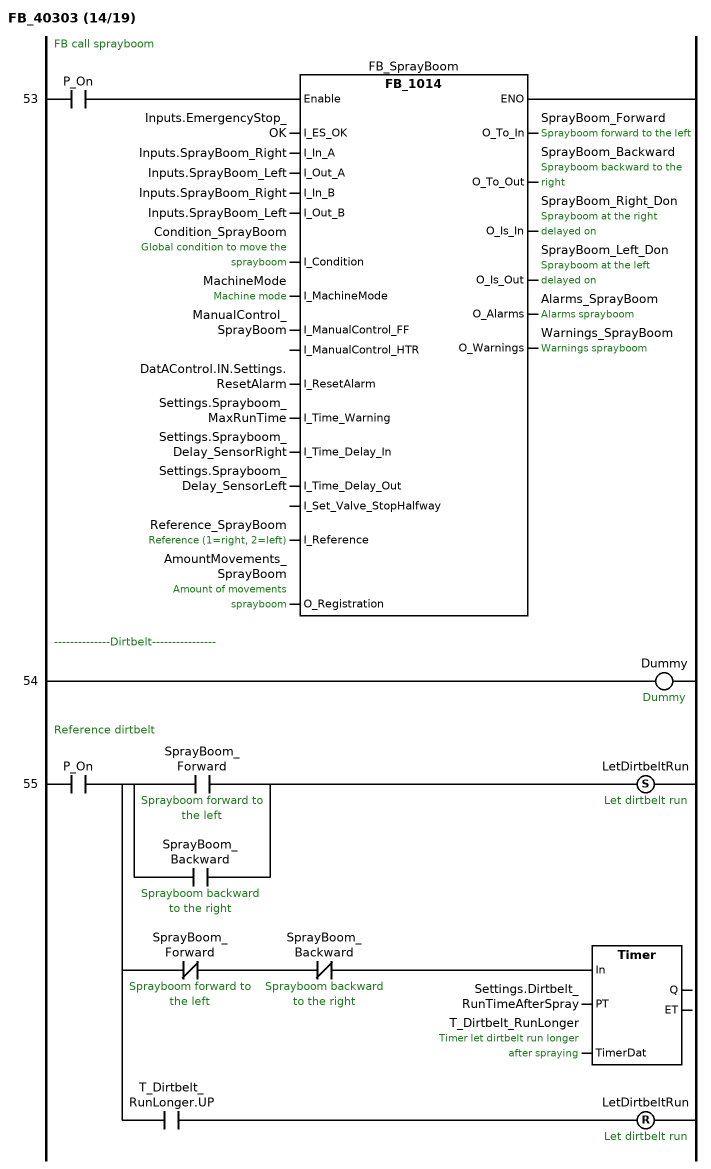
(* [picture p198: FB_40303, rungs 53-55] *)
(* Rung 53: FB call sprayboom *)
FB_SprayBoom(Enable := P_On, I_ES_OK := Inputs.EmergencyStop_OK, I_In_A := Inputs.SprayBoom_Right, I_Out_A := Inputs.SprayBoom_Left, I_In_B := Inputs.SprayBoom_Right, I_Out_B := Inputs.SprayBoom_Left, I_Condition := Condition_SprayBoom, I_MachineMode := MachineMode, I_ManualControl_FF := ManualControl_SprayBoom, I_ResetAlarm := DatAControl.IN.Settings.ResetAlarm, I_Time_Warning := Settings.Sprayboom_MaxRunTime, I_Time_Delay_In := Settings.Sprayboom_Delay_SensorRight, I_Time_Delay_Out := Settings.Sprayboom_Delay_SensorLeft, I_Reference := Reference_SprayBoom, O_Registration := AmountMovements_SprayBoom, O_To_In => SprayBoom_Forward, O_To_Out => SprayBoom_Backward, O_Is_In => SprayBoom_Right_Don, O_Is_Out => SprayBoom_Left_Don, O_Alarms => Alarms_SprayBoom, O_Warnings => Warnings_SprayBoom);
(* Rung 54: --------------Dirtbelt---------------- *)
Dummy := TRUE;
(* Rung 55: Reference dirtbelt *)
IF P_On AND (SprayBoom_Forward OR SprayBoom_Backward) THEN LetDirtbeltRun := TRUE; END_IF;
_t18 := Timer(In := P_On AND NOT SprayBoom_Forward AND NOT SprayBoom_Backward, PT := Settings.Dirtbelt_RunTimeAfterSpray, TimerDat := T_Dirtbelt_RunLonger);
IF P_On AND T_Dirtbelt_RunLonger.UP THEN LetDirtbeltRun := FALSE; END_IF;

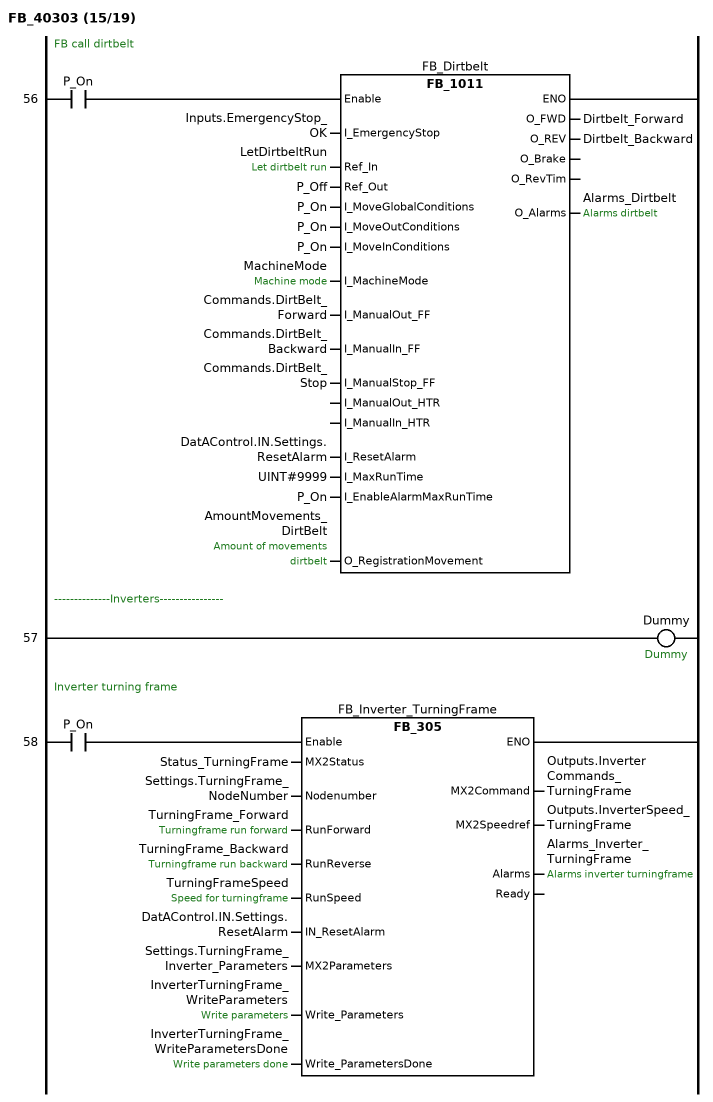
(* Rung 56: FB call dirtbelt *)
FB_Dirtbelt(Enable := P_On, I_EmergencyStop := Inputs.EmergencyStop_OK, Ref_In := LetDirtbeltRun, Ref_Out := P_Off, I_MoveGlobalConditions := P_On, I_MoveOutConditions := P_On, I_MoveInConditions := P_On, I_MachineMode := MachineMode, I_ManualOut_FF := Commands.DirtBelt_Forward, I_ManualIn_FF := Commands.DirtBelt_Backward, I_ManualStop_FF := Commands.DirtBelt_Stop, I_ResetAlarm := DatAControl.IN.Settings.ResetAlarm, I_MaxRunTime := UINT#9999, I_EnableAlarmMaxRunTime := P_On, O_RegistrationMovement := AmountMovements_DirtBelt, O_FWD => Dirtbelt_Forward, O_REV => Dirtbelt_Backward, O_Alarms => Alarms_Dirtbelt);
(* Rung 57: --------------Inverters---------------- *)
Dummy := TRUE;
(* Rung 58: Inverter turning frame *)
FB_Inverter_TurningFrame(Enable := P_On, MX2Status := Status_TurningFrame, Nodenumber := Settings.TurningFrame_NodeNumber, RunForward := TurningFrame_Forward, RunReverse := TurningFrame_Backward, RunSpeed := TurningFrameSpeed, IN_ResetAlarm := DatAControl.IN.Settings.ResetAlarm, MX2Parameters := Settings.TurningFrame_Inverter_Parameters, Write_Parameters := InverterTurningFrame_WriteParameters, Write_ParametersDone := InverterTurningFrame_WriteParametersDone, MX2Command => Outputs.InverterCommands_TurningFrame, MX2Speedref => Outputs.InverterSpeed_TurningFrame, Alarms => Alarms_Inverter_TurningFrame);

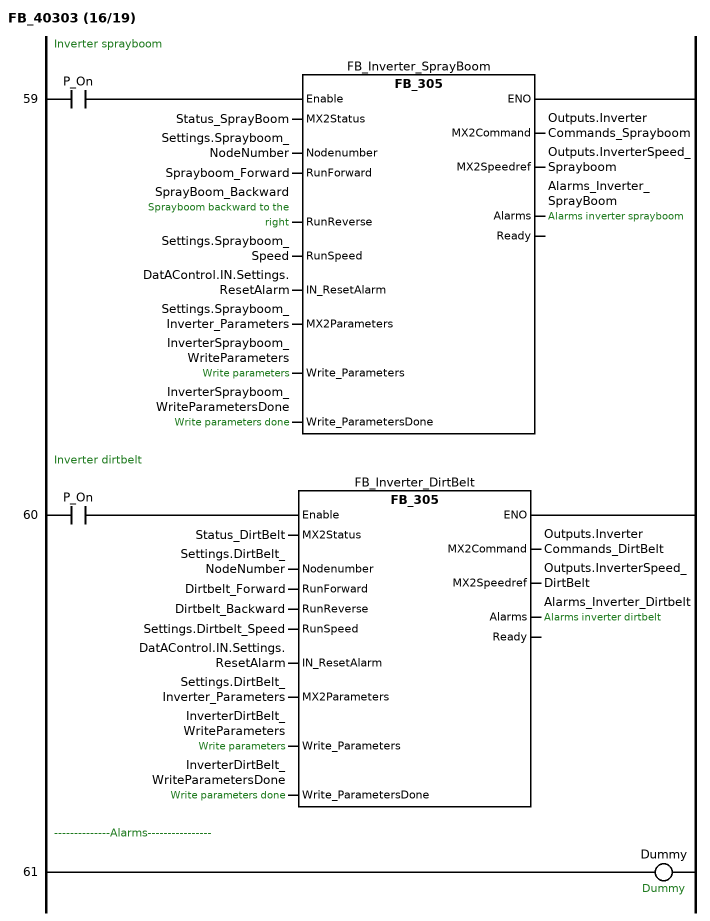
(* Rung 59: Inverter sprayboom *)
FB_Inverter_SprayBoom(Enable := P_On, MX2Status := Status_SprayBoom, Nodenumber := Settings.Sprayboom_NodeNumber, RunForward := Sprayboom_Forward, RunReverse := SprayBoom_Backward, RunSpeed := Settings.Sprayboom_Speed, IN_ResetAlarm := DatAControl.IN.Settings.ResetAlarm, MX2Parameters := Settings.Sprayboom_Inverter_Parameters, Write_Parameters := InverterSprayboom_WriteParameters, Write_ParametersDone := InverterSprayboom_WriteParametersDone, MX2Command => Outputs.InverterCommands_Sprayboom, MX2Speedref => Outputs.InverterSpeed_Sprayboom, Alarms => Alarms_Inverter_SprayBoom);
(* Rung 60: Inverter dirtbelt *)
FB_Inverter_DirtBelt(Enable := P_On, MX2Status := Status_DirtBelt, Nodenumber := Settings.DirtBelt_NodeNumber, RunForward := Dirtbelt_Forward, RunReverse := Dirtbelt_Backward, RunSpeed := Settings.Dirtbelt_Speed, IN_ResetAlarm := DatAControl.IN.Settings.ResetAlarm, MX2Parameters := Settings.DirtBelt_Inverter_Parameters, Write_Parameters := InverterDirtBelt_WriteParameters, Write_ParametersDone := InverterDirtBelt_WriteParametersDone, MX2Command => Outputs.InverterCommands_DirtBelt, MX2Speedref => Outputs.InverterSpeed_DirtBelt, Alarms => Alarms_Inverter_Dirtbelt);
(* Rung 61: --------------Alarms---------------- *)
Dummy := TRUE;

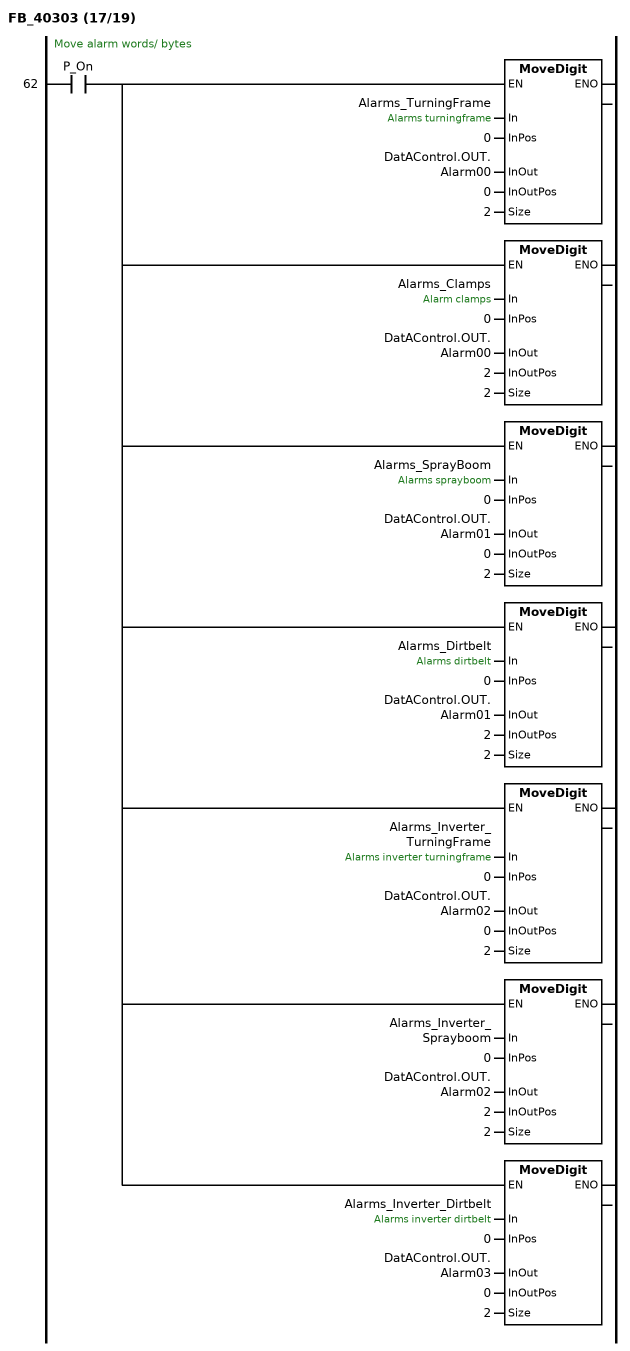
(* Rung 62: Move alarm words/ bytes *)
IF P_On THEN
    MoveDigit(In := Alarms_TurningFrame, InPos := 0, InOut := DatAControl.OUT.Alarm00, InOutPos := 0, Size := 2);
    MoveDigit(In := Alarms_Clamps, InPos := 0, InOut := DatAControl.OUT.Alarm00, InOutPos := 2, Size := 2);
    MoveDigit(In := Alarms_SprayBoom, InPos := 0, InOut := DatAControl.OUT.Alarm01, InOutPos := 0, Size := 2);
    MoveDigit(In := Alarms_Dirtbelt, InPos := 0, InOut := DatAControl.OUT.Alarm01, InOutPos := 2, Size := 2);
    MoveDigit(In := Alarms_Inverter_TurningFrame, InPos := 0, InOut := DatAControl.OUT.Alarm02, InOutPos := 0, Size := 2);
    MoveDigit(In := Alarms_Inverter_Sprayboom, InPos := 0, InOut := DatAControl.OUT.Alarm02, InOutPos := 2, Size := 2);
    MoveDigit(In := Alarms_Inverter_Dirtbelt, InPos := 0, InOut := DatAControl.OUT.Alarm03, InOutPos := 0, Size := 2);
END_IF;

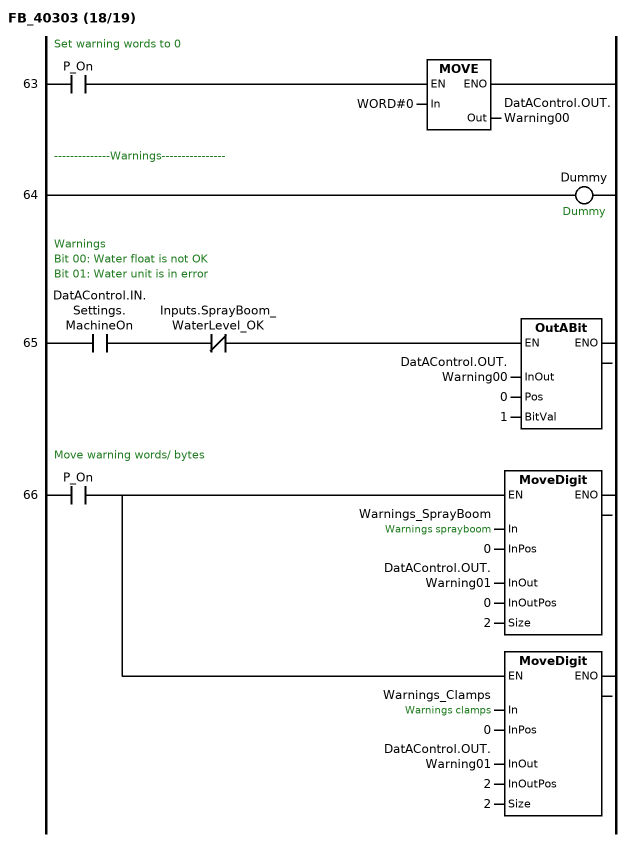
(* Rung 63: Set warning words to 0 *)
IF P_On THEN DatAControl.OUT.Warning00 := WORD#0; END_IF;
(* Rung 64: --------------Warnings---------------- *)
Dummy := TRUE;
(* Rung 65: Warnings / Bit 00: Water float is not OK / Bit 01: Water unit is in error *)
IF DatAControl.IN.Settings.MachineOn AND NOT Inputs.SprayBoom_WaterLevel_OK THEN
    OutABit(InOut := DatAControl.OUT.Warning00, Pos := 0, BitVal := 1);
END_IF;
(* Rung 66: Move warning words/ bytes *)
IF P_On THEN
    MoveDigit(In := Warnings_SprayBoom, InPos := 0, InOut := DatAControl.OUT.Warning01, InOutPos := 0, Size := 2);
    MoveDigit(In := Warnings_Clamps, InPos := 0, InOut := DatAControl.OUT.Warning01, InOutPos := 2, Size := 2);
END_IF;

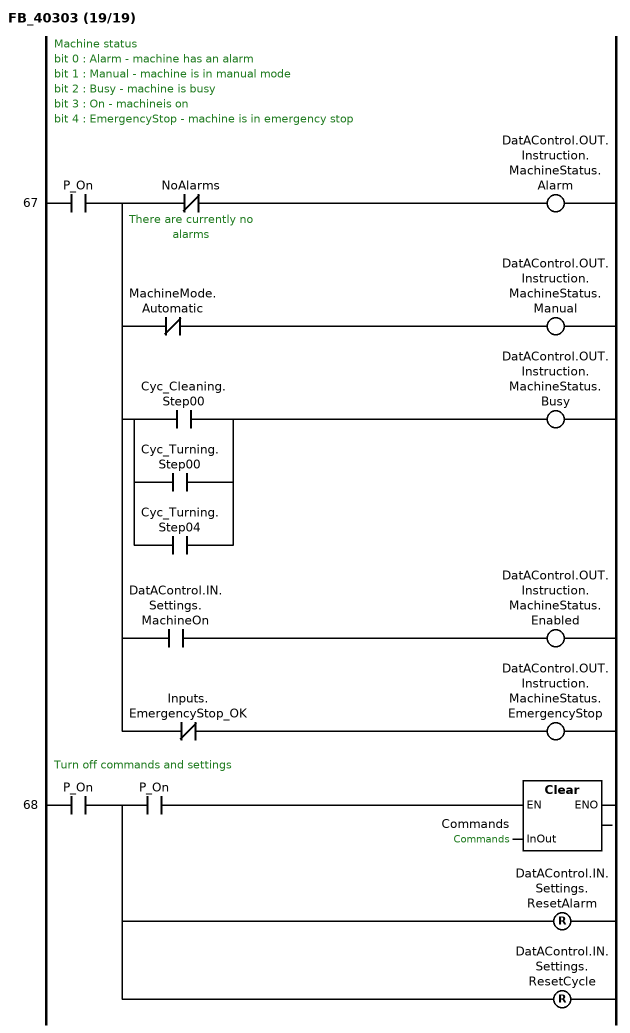
(* Rung 67: Machine status / bit 0 : Alarm - machine has an alarm / bit 1 : Manual - machine is in manual mode / bit 2 : Busy - machine is busy / bit 3 : On - machineis on / bit 4 : EmergencyStop - machine is in emergency stop *)
DatAControl.OUT.Instruction.MachineStatus.Alarm := P_On AND NOT NoAlarms;
DatAControl.OUT.Instruction.MachineStatus.Manual := P_On AND NOT MachineMode.Automatic;
DatAControl.OUT.Instruction.MachineStatus.Busy := P_On AND (Cyc_Cleaning.Step00 OR Cyc_Turning.Step00 OR Cyc_Turning.Step04);
DatAControl.OUT.Instruction.MachineStatus.Enabled := P_On AND DatAControl.IN.Settings.MachineOn;
DatAControl.OUT.Instruction.MachineStatus.EmergencyStop := P_On AND NOT Inputs.EmergencyStop_OK;
(* Rung 68: Turn off commands and settings *)
IF P_On AND P_On THEN Clear(InOut := Commands); END_IF;
IF P_On THEN
    DatAControl.IN.Settings.ResetAlarm := FALSE;
    DatAControl.IN.Settings.ResetCycle := FALSE;
END_IF;
END_FUNCTION_BLOCK

FUNCTION_BLOCK FB_1017
(* Valve movement bi-directional with 4 sensors for in detection and 4 sensors for out detection *)
VAR
    Reference_In : BOOL;  (* Reference is in *)
    Reference_Out : BOOL;  (* Reference is out *)
    Manual_In : BOOL;  (* ManualControl in *)
    Manual_Out : BOOL;  (* ManualControl out *)
    Desired_To_Out : BOOL;  (* Movement desired to Out *)
    Desired_To_In : BOOL;  (* Movement desired to In *)
    Sensor_Out_A : BOOL;  (* Sensor out side A *)
    Sensor_Out_A_Don : BOOL;  (* Sensor out side A delayed *)
    Sensor_In_A : BOOL;  (* Sensor in side A *)
    Sensor_In_A_Don : BOOL;  (* Sensor in side A delayed *)
    ManualControl : FB_303;
    Actuator_is_Out : BOOL;  (* Actuator is out *)
    Actuator_is_In : BOOL;  (* Actuator is in *)
    Input_Out_A : FB_101;
    Input_In_A : FB_101;
    Alarm_SensorTogether_A : FB_502;
    Alarm_MaxRunTime : BOOL;  (* Alarm maximum runtime actuator *)
    Alarm_Switch_Together_A : BOOL;  (* Alarm switches switched together side A *)
    Input_Out_B : FB_101;
    Sensor_Out_B : BOOL;  (* Sensor out side B *)
    Sensor_Out_B_Don : BOOL;  (* Sensor out side B delayed *)
    Input_In_B : FB_101;
    Sensor_In_B : BOOL;  (* Sensor in side B *)
    Sensor_In_B_Don : BOOL;  (* Sensor in side B delayed *)
    Alarm_SensorTogether_B : FB_502;
    Alarm_Switch_Together_B : BOOL;  (* Alarm switches switched together side B *)
    T_Warn_Out : _sTimer;
    T_Warn_In : _sTimer;
    ReversalProtection_A : FB_201;
    ReversalProtection_B : FB_201;
    NotRunning_A : BOOL;
    NotRunning_B : BOOL;
END_VAR
VAR_INPUT
    Enable : BOOL;
    I_ES_OK : BOOL;  (* IN: EmergencyStop OK *)
    I_In_A : BOOL;  (* IN: Sensor in side A *)
    I_Out_A : BOOL;  (* IN: Sensor out side A *)
    I_In_B : BOOL;  (* IN: Sensor in side B *)
    I_Out_B : BOOL;  (* IN: Sensor out side B *)
    I_Condition : BOOL;  (* IN: Global condition to move *)
    I_MachineMode : ST_MachineMode;  (* IN: Machine mode *)
    I_ManualControl : ST_ManualControl_Actuator;  (* IN: Manual control *)
    I_ResetAlarm : BOOL;  (* IN: Reset alarm *)
    I_Reference : UINT;  (* IN: Reference (1 = In, 2 = Out *)
    I_Time_Warning : UINT;  (* IN: Time for warnings 'does not reach end switch' *)
    I_Time_Delay_In : UINT;  (* IN: Time delay on in sensor *)
    I_Time_Delay_Out : UINT;  (* IN: Time delay on out sensor *)
END_VAR
VAR_OUTPUT
    O_To_In_A : BOOL;  (* OUT: Valve in A *)
    O_To_Out_A : BOOL;  (* OUT: Valve out A *)
    O_To_In_B : BOOL;  (* OUT: Valve in B *)
    O_To_Out_B : BOOL;  (* OUT: Valve out B *)
    O_Is_In : BOOL;  (* OUT: Unit is in *)
    O_Is_Out : BOOL;  (* OUT: Unit is out *)
    O_Alarms : BYTE;  (* OUT: Alarms *)
    O_Warnings : BYTE;  (* OUT: Warnings *)
END_VAR
VAR_IN_OUT
    O_Registration : UDINT;  (* OUT: Total amount of movements *)
END_VAR
VAR
    _t1 : BOOL;
    _t2 : BOOL;
    _e3 : R_TRIG;
    _e4 : R_TRIG;
END_VAR
(* ladder, written here as Structured Text *)

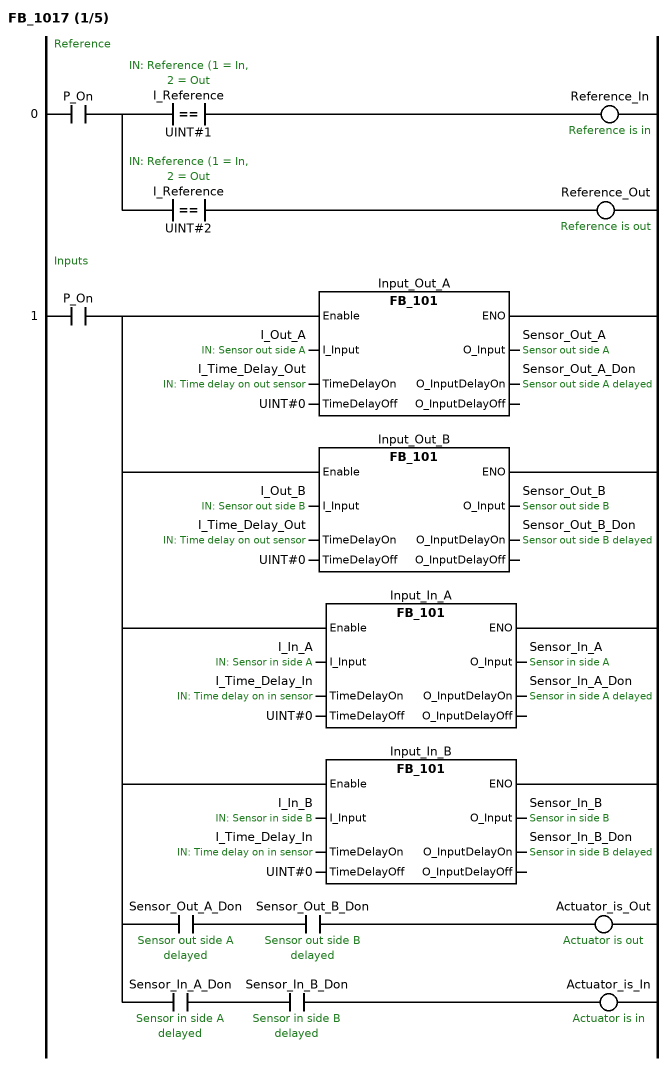
(* Rung 0: Reference *)
Reference_In := P_On AND (I_Reference = UINT#1);
Reference_Out := P_On AND (I_Reference = UINT#2);
(* Rung 1: Inputs *)
Input_Out_A(Enable := P_On, I_Input := I_Out_A, TimeDelayOn := I_Time_Delay_Out, TimeDelayOff := UINT#0, O_Input => Sensor_Out_A, O_InputDelayOn => Sensor_Out_A_Don);
Input_Out_B(Enable := P_On, I_Input := I_Out_B, TimeDelayOn := I_Time_Delay_Out, TimeDelayOff := UINT#0, O_Input => Sensor_Out_B, O_InputDelayOn => Sensor_Out_B_Don);
Input_In_A(Enable := P_On, I_Input := I_In_A, TimeDelayOn := I_Time_Delay_In, TimeDelayOff := UINT#0, O_Input => Sensor_In_A, O_InputDelayOn => Sensor_In_A_Don);
Input_In_B(Enable := P_On, I_Input := I_In_B, TimeDelayOn := I_Time_Delay_In, TimeDelayOff := UINT#0, O_Input => Sensor_In_B, O_InputDelayOn => Sensor_In_B_Don);
Actuator_is_Out := P_On AND Sensor_Out_A_Don AND Sensor_Out_B_Don;
Actuator_is_In := P_On AND Sensor_In_A_Don AND Sensor_In_B_Don;

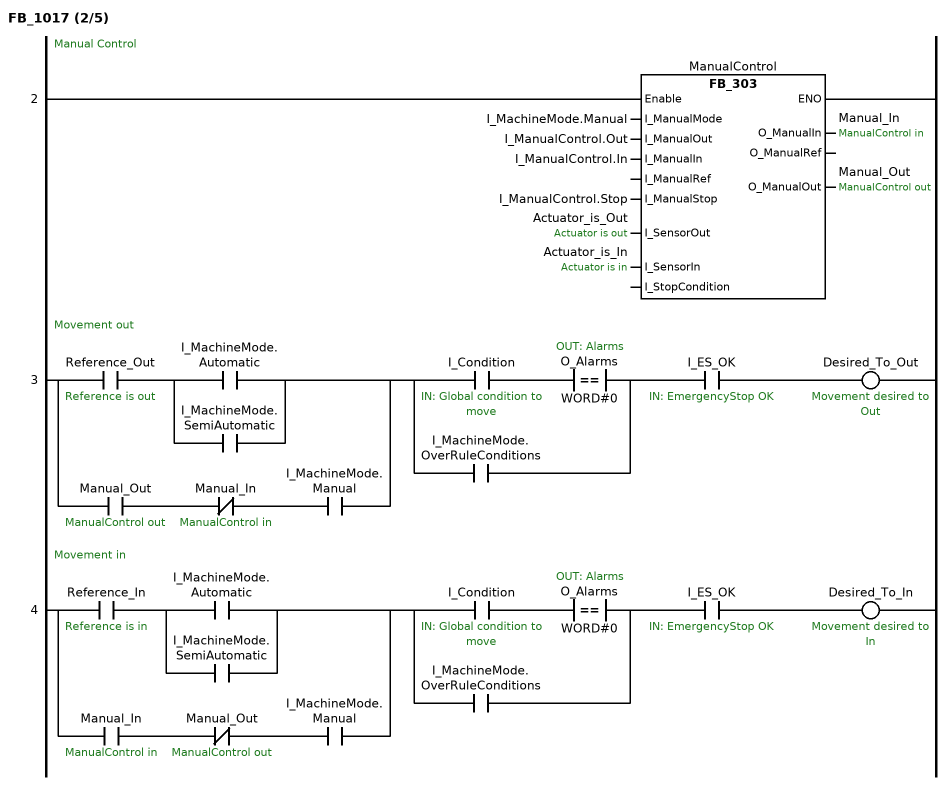
(* Rung 2: Manual Control *)
ManualControl(Enable := TRUE, I_ManualMode := I_MachineMode.Manual, I_ManualOut := I_ManualControl.Out, I_ManualIn := I_ManualControl.In, I_ManualStop := I_ManualControl.Stop, I_SensorOut := Actuator_is_Out, I_SensorIn := Actuator_is_In, O_ManualIn => Manual_In, O_ManualOut => Manual_Out);
(* Rung 3: Movement out *)
Desired_To_Out := ((Reference_Out AND (I_MachineMode.Automatic OR I_MachineMode.SemiAutomatic)) OR (Manual_Out AND NOT Manual_In AND I_MachineMode.Manual)) AND ((I_Condition AND (O_Alarms = WORD#0)) OR I_MachineMode.OverRuleConditions) AND I_ES_OK;
(* Rung 4: Movement in *)
Desired_To_In := ((Reference_In AND (I_MachineMode.Automatic OR I_MachineMode.SemiAutomatic)) OR (Manual_In AND NOT Manual_Out AND I_MachineMode.Manual)) AND ((I_Condition AND (O_Alarms = WORD#0)) OR I_MachineMode.OverRuleConditions) AND I_ES_OK;

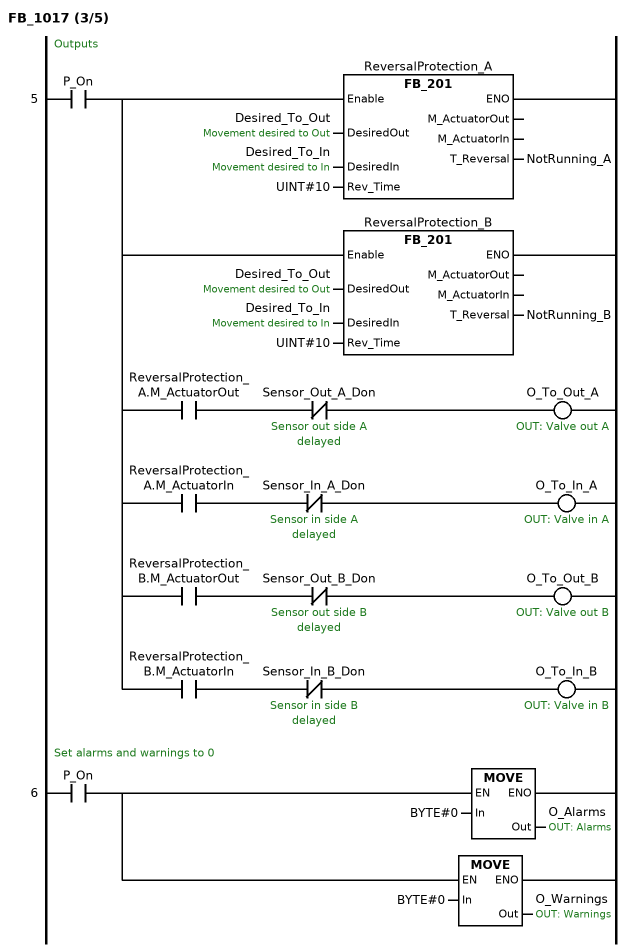
(* Rung 5: Outputs *)
ReversalProtection_A(Enable := P_On, DesiredOut := Desired_To_Out, DesiredIn := Desired_To_In, Rev_Time := UINT#10, T_Reversal => NotRunning_A);
ReversalProtection_B(Enable := P_On, DesiredOut := Desired_To_Out, DesiredIn := Desired_To_In, Rev_Time := UINT#10, T_Reversal => NotRunning_B);
O_To_Out_A := P_On AND ReversalProtection_A.M_ActuatorOut AND NOT Sensor_Out_A_Don;
O_To_In_A := P_On AND ReversalProtection_A.M_ActuatorIn AND NOT Sensor_In_A_Don;
O_To_Out_B := P_On AND ReversalProtection_B.M_ActuatorOut AND NOT Sensor_Out_B_Don;
O_To_In_B := P_On AND ReversalProtection_B.M_ActuatorIn AND NOT Sensor_In_B_Don;
(* Rung 6: Set alarms and warnings to 0 *)
IF P_On THEN
    O_Alarms := BYTE#0;
    O_Warnings := BYTE#0;
END_IF;

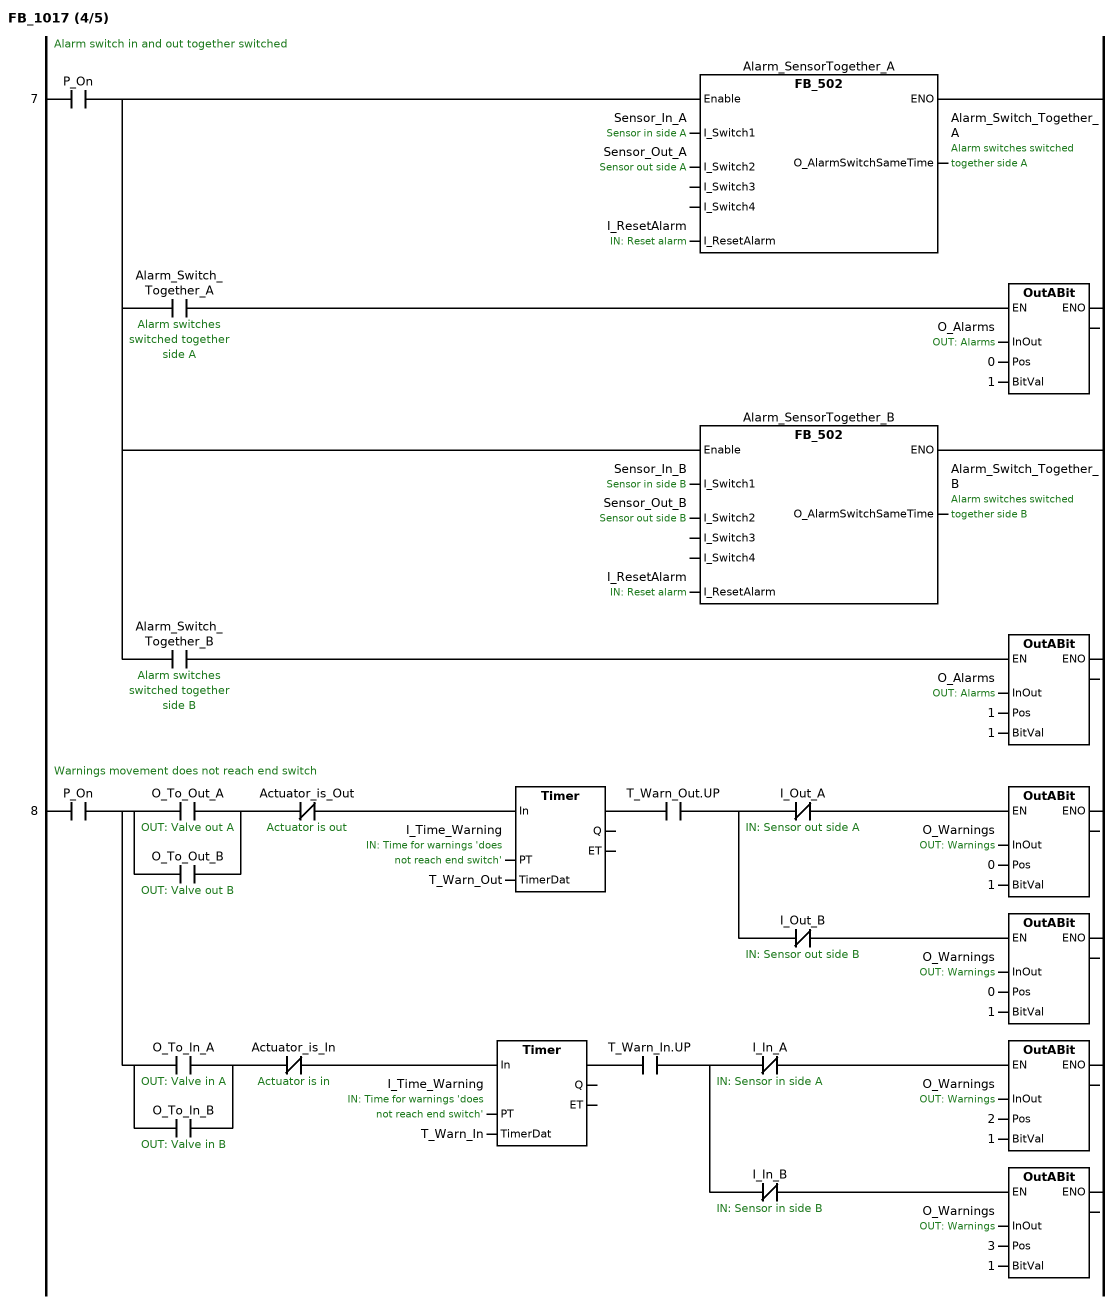
(* Rung 7: Alarm switch in and out together switched *)
Alarm_SensorTogether_A(Enable := P_On, I_Switch1 := Sensor_In_A, I_Switch2 := Sensor_Out_A, I_ResetAlarm := I_ResetAlarm, O_AlarmSwitchSameTime => Alarm_Switch_Together_A);
IF P_On AND Alarm_Switch_Together_A THEN OutABit(InOut := O_Alarms, Pos := 0, BitVal := 1); END_IF;
Alarm_SensorTogether_B(Enable := P_On, I_Switch1 := Sensor_In_B, I_Switch2 := Sensor_Out_B, I_ResetAlarm := I_ResetAlarm, O_AlarmSwitchSameTime => Alarm_Switch_Together_B);
IF P_On AND Alarm_Switch_Together_B THEN OutABit(InOut := O_Alarms, Pos := 1, BitVal := 1); END_IF;
(* Rung 8: Warnings movement does not reach end switch *)
_t1 := Timer(In := P_On AND (O_To_Out_A OR O_To_Out_B) AND NOT Actuator_is_Out, PT := I_Time_Warning, TimerDat := T_Warn_Out);
IF _t1 AND T_Warn_Out.UP AND NOT I_Out_A THEN OutABit(InOut := O_Warnings, Pos := 0, BitVal := 1); END_IF;
IF _t1 AND T_Warn_Out.UP AND NOT I_Out_B THEN OutABit(InOut := O_Warnings, Pos := 0, BitVal := 1); END_IF;
_t2 := Timer(In := P_On AND (O_To_In_A OR O_To_In_B) AND NOT Actuator_is_In, PT := I_Time_Warning, TimerDat := T_Warn_In);
IF _t2 AND T_Warn_In.UP AND NOT I_In_A THEN OutABit(InOut := O_Warnings, Pos := 2, BitVal := 1); END_IF;
IF _t2 AND T_Warn_In.UP AND NOT I_In_B THEN OutABit(InOut := O_Warnings, Pos := 3, BitVal := 1); END_IF;

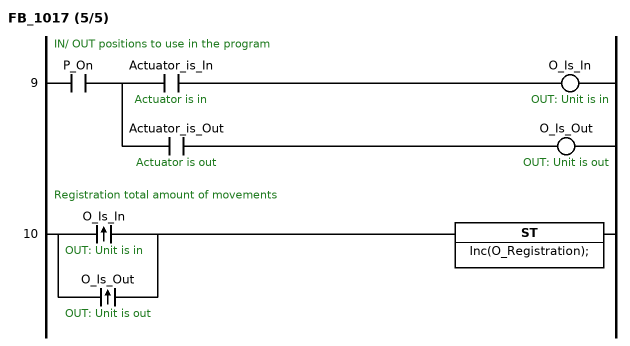
(* Rung 9: IN/ OUT positions to use in the program *)
O_Is_In := P_On AND Actuator_is_In;
O_Is_Out := P_On AND Actuator_is_Out;
(* Rung 10: Registration total amount of movements *)
_e3(CLK := O_Is_In);
_e4(CLK := O_Is_Out);
IF _e3.Q OR _e4.Q THEN
    Inc(O_Registration);
    	
END_IF;
END_FUNCTION_BLOCK

FUNCTION_BLOCK FB_1018
VAR
    Reference_In : BOOL;  (* Reference is in *)
    Reference_Middle : BOOL;  (* Reference is middle *)
    Reference_Out : BOOL;  (* Reference is out *)
    Input_In : FB_101;
    Input_Out : FB_101;
    Input_Middle : FB_101;
    SensorIn_Don : BOOL;  (* Sensor in delayed on *)
    SensorOut_Don : BOOL;  (* Sensor out delayed on *)
    SensorMiddle_Don : BOOL;  (* Sensor middle delayed on *)
    ManualControl : FB_303;
    Manual_To_Out : BOOL;  (* Manual to the out *)
    Manual_To_In : BOOL;  (* Manual to the in *)
    Desired_To_Out : BOOL;  (* Desired to go to the out *)
    Desired_To_In : BOOL;  (* Desired to go to the in *)
END_VAR
VAR RETAIN
    Position : BOOL;  (* Position (0=in of middle position, 1=out of middle position) *)
END_VAR
VAR
    ReversalProtection : FB_201;
    NotRunning : BOOL;
    FB_Alarm_Runtime : FB_501;
    Alarm_Runtime : BOOL;
    FB_Alarm_MultipleSwithches : FB_502;
    Alarm_MultipleSwitches : BOOL;
    Alarm_Direction : BOOL;
    Alarm_NoPulses : BOOL;
    Alarm_SensorInWrong : BOOL;
    Alarm_SensorOutWrong : BOOL;
    Alarm_SensorMiddleWrong : BOOL;
    T_HighSpeed_Out : _sTimer;  (* Timer high speed out *)
    T_HighSpeed_In : _sTimer;  (* Timer high speed in *)
END_VAR
VAR_INPUT
    I_Enable : BOOL;
    I_ES_OK : BOOL;  (* IN: EmergencyStop OK *)
    I_In : BOOL;  (* IN: In *)
    I_Middle : BOOL;  (* IN:  Middle *)
    I_Out : BOOL;  (* IN: Out *)
    I_Delay_In : UINT;  (* IN: Time delay on sensor in *)
    I_Delay_Middle : UINT;  (* IN: Time delay on sensor middle *)
    I_Delay_Out : UINT;  (* IN: Time delay on sensor out *)
    I_Conditions_In : BOOL;  (* IN: Conditions move in *)
    I_Conditions_Out : BOOL;  (* IN: Conditions move out *)
    I_MachineMode : ST_MachineMode;  (* IN: Machine mode *)
    I_ManualControl : ST_ManualControl_Actuator;
    I_ResetAlarm : BOOL;  (* IN: Reset alarm *)
    I_Reference : UINT;  (* IN: Reference (1=in, 2=middle, 3=out) *)
    I_MINSpeed : UINT;  (* Minimum speed *)
    I_MAXSpeed : UINT;  (* Maximum speed *)
    I_MaxRunTime : UINT;  (* IN: Maximum runtime *)
    I_Time_HighSpeedIn : UINT;  (* IN: Time movement high speed in *)
    I_Time_HighSpeedOut : UINT;  (* IN: Time movement high speed out *)
END_VAR
VAR_OUTPUT
    O_To_In : BOOL;  (* OUT: In *)
    O_To_Out : BOOL;  (* OUT: Out *)
    O_Is_In : BOOL;  (* OUT: Unit is in *)
    O_Is_Middle : BOOL;  (* OUT: Unit is middle *)
    O_Is_Out : BOOL;  (* OUT: Unit is out *)
    O_Brake : BOOL;  (* OUT: Brake *)
    O_Speed : UINT;  (* OUT: Desired speed *)
END_VAR
VAR_OUTPUT RETAIN
    O_Alarms : BYTE;  (* OUT: Alarms *)
END_VAR
VAR_IN_OUT
    O_Registration : UDINT;  (* OUT: Total amount of movements *)
END_VAR
VAR
    _e1 : F_TRIG;
    _e2 : F_TRIG;
    _t3 : BOOL;
    _t4 : BOOL;
    _e5 : R_TRIG;
    _e6 : R_TRIG;
END_VAR
(* ladder, written here as Structured Text *)

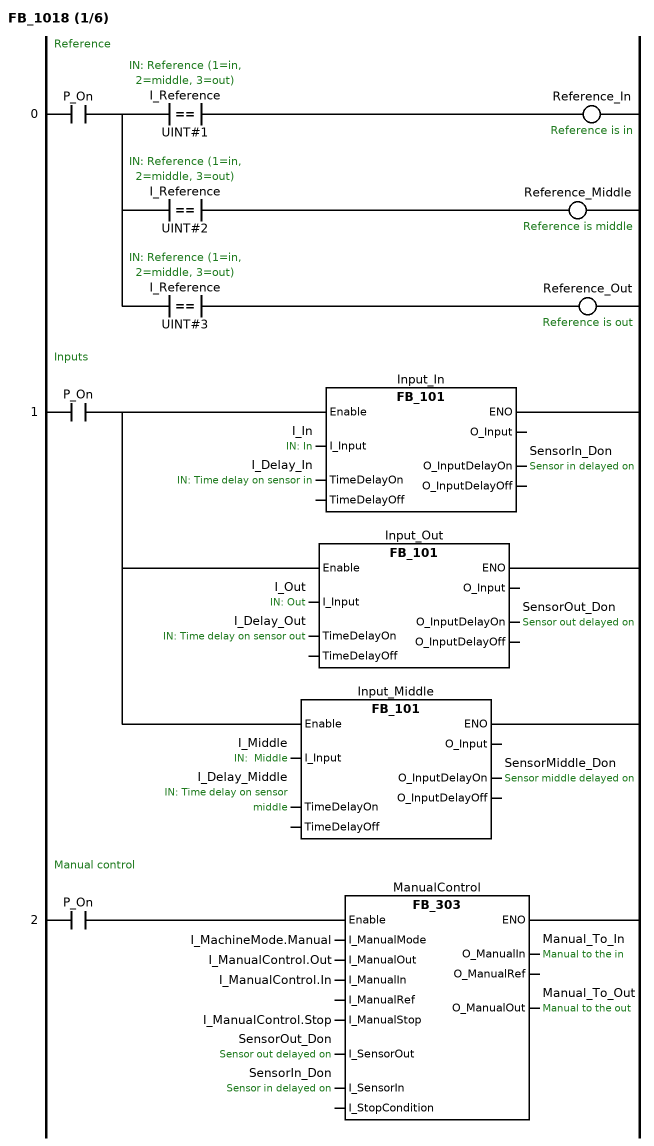
(* Rung 0: Reference *)
Reference_In := P_On AND (I_Reference = UINT#1);
Reference_Middle := P_On AND (I_Reference = UINT#2);
Reference_Out := P_On AND (I_Reference = UINT#3);
(* Rung 1: Inputs *)
Input_In(Enable := P_On, I_Input := I_In, TimeDelayOn := I_Delay_In, O_InputDelayOn => SensorIn_Don);
Input_Out(Enable := P_On, I_Input := I_Out, TimeDelayOn := I_Delay_Out, O_InputDelayOn => SensorOut_Don);
Input_Middle(Enable := P_On, I_Input := I_Middle, TimeDelayOn := I_Delay_Middle, O_InputDelayOn => SensorMiddle_Don);
(* Rung 2: Manual control *)
ManualControl(Enable := P_On, I_ManualMode := I_MachineMode.Manual, I_ManualOut := I_ManualControl.Out, I_ManualIn := I_ManualControl.In, I_ManualStop := I_ManualControl.Stop, I_SensorOut := SensorOut_Don, I_SensorIn := SensorIn_Don, O_ManualIn => Manual_To_In, O_ManualOut => Manual_To_Out);

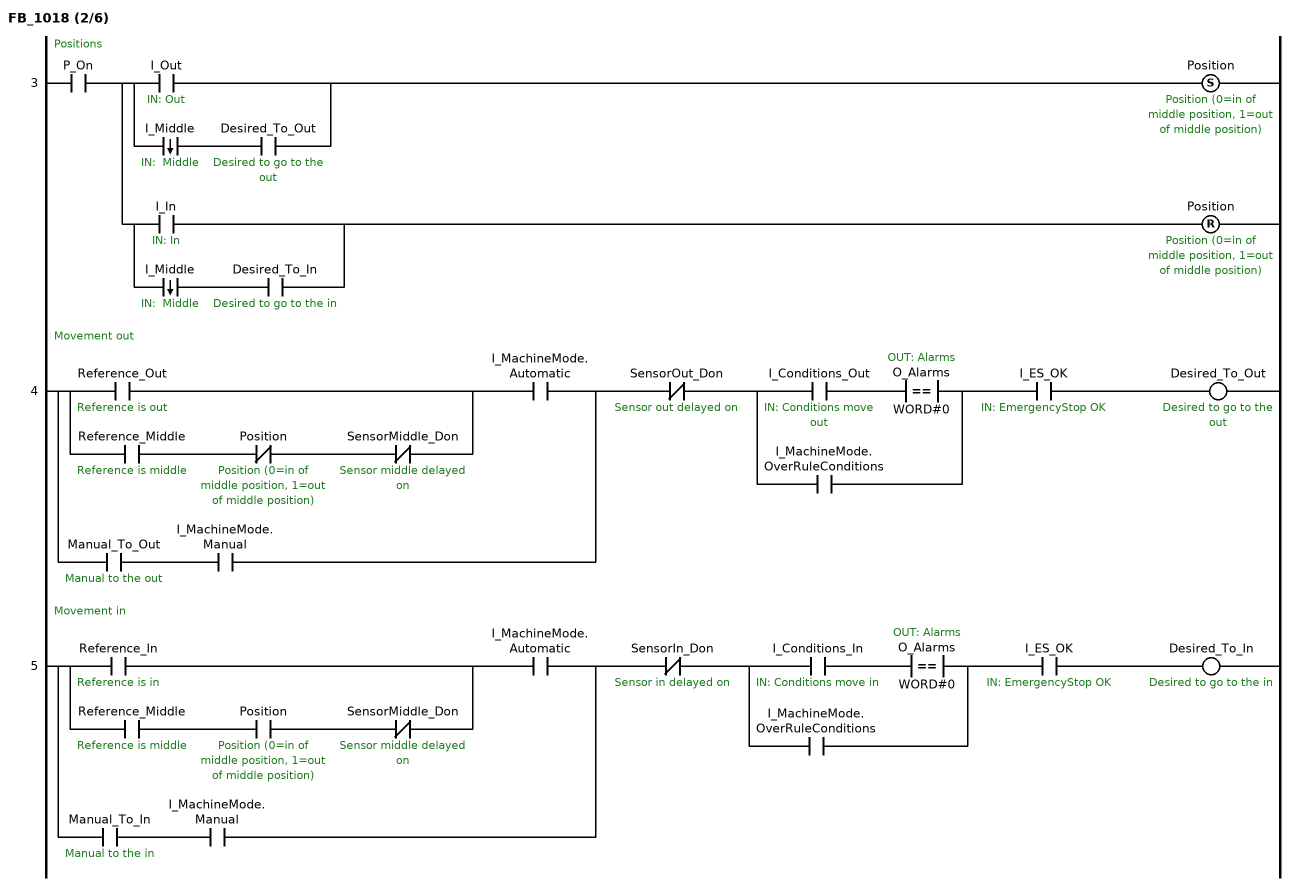
(* Rung 3: Positions *)
_e1(CLK := I_Middle);
IF P_On AND (I_Out OR (_e1.Q AND Desired_To_Out)) THEN Position := TRUE; END_IF;
_e2(CLK := I_Middle);
IF P_On AND (I_In OR (_e2.Q AND Desired_To_In)) THEN Position := FALSE; END_IF;
(* Rung 4: Movement out *)
Desired_To_Out := (((Reference_Out OR (Reference_Middle AND NOT Position AND NOT SensorMiddle_Don)) AND I_MachineMode.Automatic) OR (Manual_To_Out AND I_MachineMode.Manual)) AND NOT SensorOut_Don AND ((I_Conditions_Out AND (O_Alarms = WORD#0)) OR I_MachineMode.OverRuleConditions) AND I_ES_OK;
(* Rung 5: Movement in *)
Desired_To_In := (((Reference_In OR (Reference_Middle AND Position AND NOT SensorMiddle_Don)) AND I_MachineMode.Automatic) OR (Manual_To_In AND I_MachineMode.Manual)) AND NOT SensorIn_Don AND ((I_Conditions_In AND (O_Alarms = WORD#0)) OR I_MachineMode.OverRuleConditions) AND I_ES_OK;

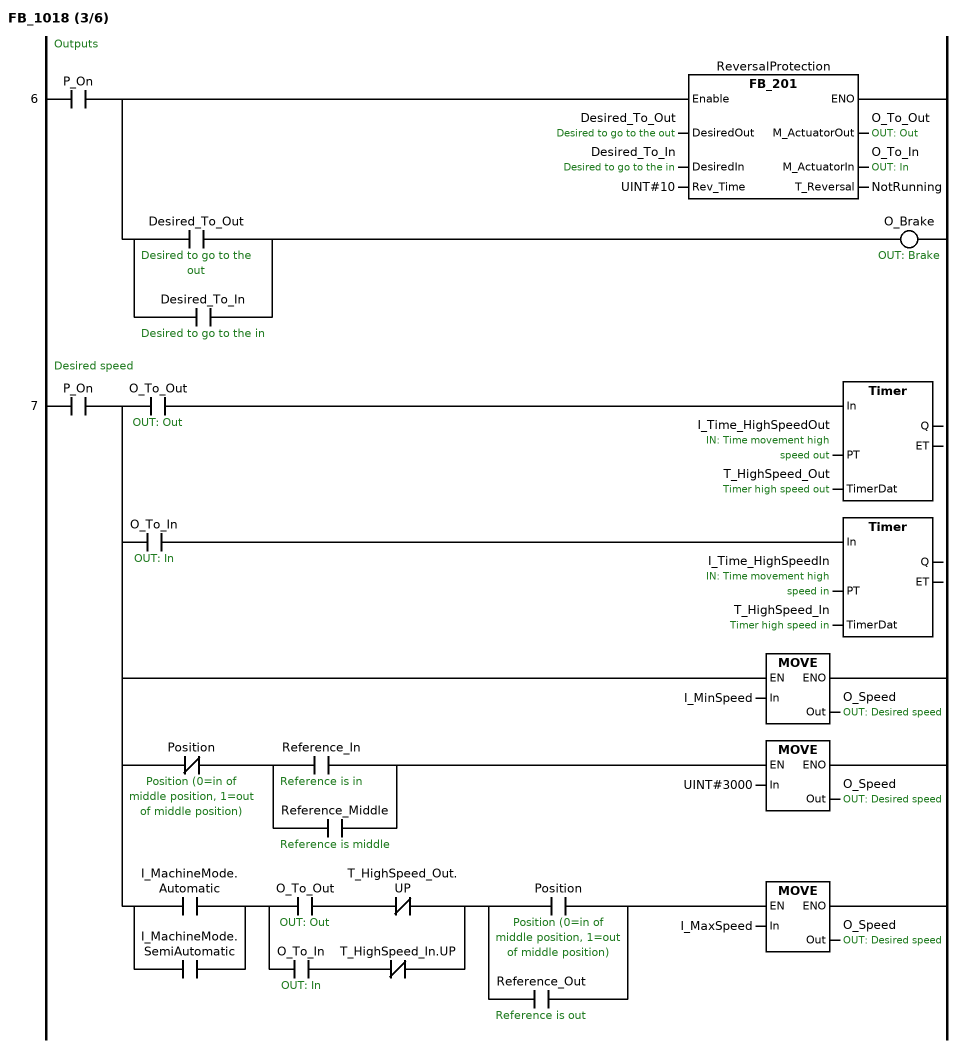
(* Rung 6: Outputs *)
ReversalProtection(Enable := P_On, DesiredOut := Desired_To_Out, DesiredIn := Desired_To_In, Rev_Time := UINT#10, M_ActuatorOut => O_To_Out, M_ActuatorIn => O_To_In, T_Reversal => NotRunning);
O_Brake := P_On AND (Desired_To_Out OR Desired_To_In);
(* Rung 7: Desired speed *)
_t3 := Timer(In := P_On AND O_To_Out, PT := I_Time_HighSpeedOut, TimerDat := T_HighSpeed_Out);
_t4 := Timer(In := P_On AND O_To_In, PT := I_Time_HighSpeedIn, TimerDat := T_HighSpeed_In);
IF P_On THEN O_Speed := I_MinSpeed; END_IF;
IF P_On AND NOT Position AND (Reference_In OR Reference_Middle) THEN O_Speed := UINT#3000; END_IF;
IF P_On AND (I_MachineMode.Automatic OR I_MachineMode.SemiAutomatic) AND ((O_To_Out AND NOT T_HighSpeed_Out.UP) OR (O_To_In AND NOT T_HighSpeed_In.UP)) AND (Position OR Reference_Out) THEN
    O_Speed := I_MaxSpeed;
END_IF;

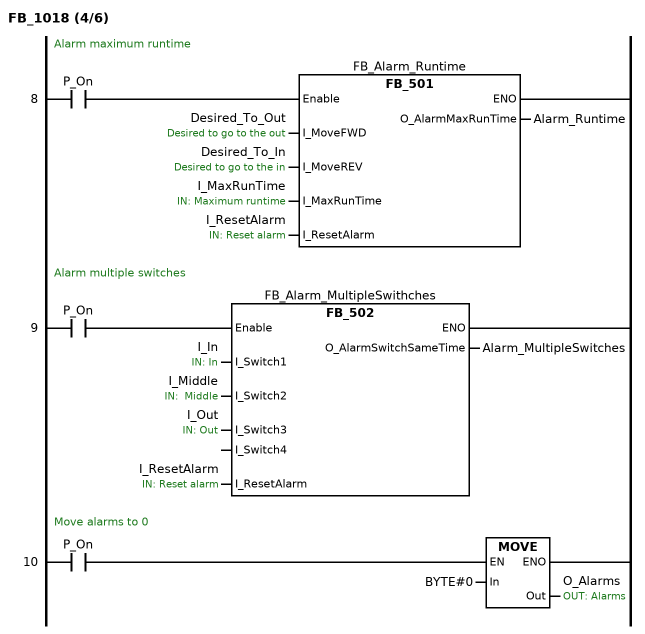
(* Rung 8: Alarm maximum runtime *)
FB_Alarm_Runtime(Enable := P_On, I_MoveFWD := Desired_To_Out, I_MoveREV := Desired_To_In, I_MaxRunTime := I_MaxRunTime, I_ResetAlarm := I_ResetAlarm, O_AlarmMaxRunTime => Alarm_Runtime);
(* Rung 9: Alarm multiple switches *)
FB_Alarm_MultipleSwithches(Enable := P_On, I_Switch1 := I_In, I_Switch2 := I_Middle, I_Switch3 := I_Out, I_ResetAlarm := I_ResetAlarm, O_AlarmSwitchSameTime => Alarm_MultipleSwitches);
(* Rung 10: Move alarms to 0 *)
IF P_On THEN O_Alarms := BYTE#0; END_IF;

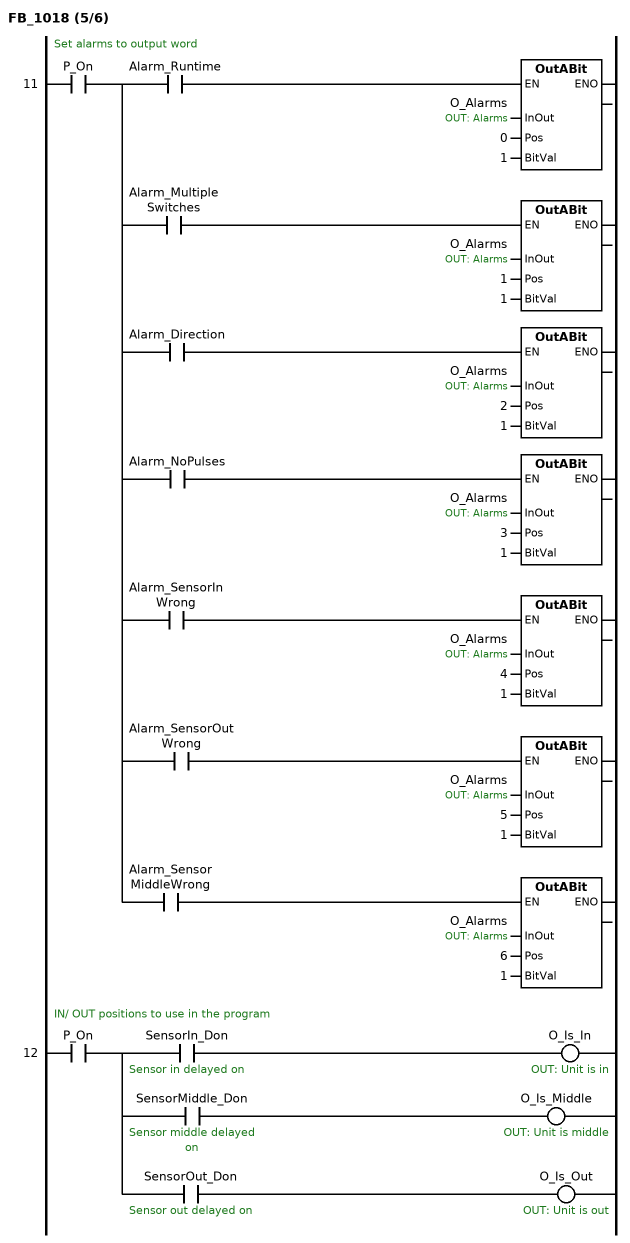
(* Rung 11: Set alarms to output word *)
IF P_On AND Alarm_Runtime THEN OutABit(InOut := O_Alarms, Pos := 0, BitVal := 1); END_IF;
IF P_On AND Alarm_MultipleSwitches THEN OutABit(InOut := O_Alarms, Pos := 1, BitVal := 1); END_IF;
IF P_On AND Alarm_Direction THEN OutABit(InOut := O_Alarms, Pos := 2, BitVal := 1); END_IF;
IF P_On AND Alarm_NoPulses THEN OutABit(InOut := O_Alarms, Pos := 3, BitVal := 1); END_IF;
IF P_On AND Alarm_SensorInWrong THEN OutABit(InOut := O_Alarms, Pos := 4, BitVal := 1); END_IF;
IF P_On AND Alarm_SensorOutWrong THEN OutABit(InOut := O_Alarms, Pos := 5, BitVal := 1); END_IF;
IF P_On AND Alarm_SensorMiddleWrong THEN OutABit(InOut := O_Alarms, Pos := 6, BitVal := 1); END_IF;
(* Rung 12: IN/ OUT positions to use in the program *)
O_Is_In := P_On AND SensorIn_Don;
O_Is_Middle := P_On AND SensorMiddle_Don;
O_Is_Out := P_On AND SensorOut_Don;

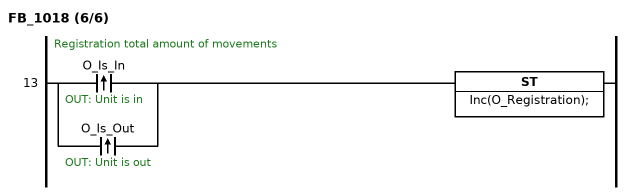
(* Rung 13: Registration total amount of movements *)
_e5(CLK := O_Is_In);
_e6(CLK := O_Is_Out);
IF _e5.Q OR _e6.Q THEN
    Inc(O_Registration);
    	
END_IF;
END_FUNCTION_BLOCK

FUNCTION_BLOCK FB_30051
VAR
    IS_TRack_201 : FB_101;
    I_Track201 : BOOL;  (* Input track 201 *)
    I_Track201DON : BOOL;  (* Input track 201 time delay on *)
    I_Track201DOFF : BOOL;  (* Input track 201 time delay off *)
    IS_Track_202 : FB_101;
    I_Track202 : BOOL;  (* input track 202 *)
    I_Track202DON : BOOL;  (* Input track 202 time delay on *)
    I_Track202DOFF : BOOL;  (* Input track 202 time delay off *)
    LS_Track_Up : FB_101;
    I_BeltUp : BOOL;  (* Input track up *)
    I_BeltUpDON : BOOL;  (* Input track up delay on *)
    LS_Track_Down : FB_101;
    I_BeltDown : BOOL;  (* Input track down *)
    I_BeltDownDON : BOOL;  (* Input track down delay on *)
    IS_Present : FB_101;
    I_Present : BOOL;  (* Input bench present *)
    I_PresentDON : BOOL;  (* Input present time delay on *)
    I_PresentDOFF : BOOL;  (* Input present delay off *)
    PB_Run_Motor : FB_101;
    I_PB_Run : BOOL;  (* Input pushbutton run motor *)
    MachineMode : ST_MachineMode;  (* Automatic Machine is automatic; SemiAutomatic Machine is semi automatic; Manual Machine is in manual *)
END_VAR
VAR RETAIN
    Cyc_Inb : ST_FB_30051_Cyc_Inbound;  (* Cycle inbound *)
    Cyc_Outb : ST_FB_30051_Cyc_Outbound;  (* Cycle outbound *)
    Cyc_Track201 : ST_FB_30051_Cyc_Track201;  (* Cycle track 201 *)
    Cyc_Track202 : ST_FB_30051_Cyc_Track202;  (* Cycle track 202 *)
END_VAR
VAR
    Instruction : FB_904;
    InstructionConditions : ST_Instruction_Conditions_Standaard;  (* Instruction conditions *)
    Start_Instruction : BOOL;  (* start instruction *)
    LoadGate : UINT;  (* Load gate *)
    UnloadGate : UINT;  (* unload gate *)
    Track_DirectionFromBuffer : BOOL;  (* Track direction from buffer *)
    Track_DirectionToBuffer : BOOL;  (* Track direction to buffer *)
    Reset_Alarm : BOOL;  (* Reset Alarm *)
    Reset_Cycle : BOOL;  (* Reset Cycle *)
    TransferOK : BOOL;  (* Transfer ok *)
    ConditionsFWD_OK : BOOL;  (* Conditions track forward ok *)
    ConditionsREV_OK : BOOL;  (* Conditions track reverse ok *)
    ConditionsGlobal_OK : BOOL;  (* Conditions global ok *)
    Track_Ref_FWD : BOOL;  (* Track reference is fwd *)
    Track_Ref_REV : BOOL;  (* Track reference is REV *)
    TrackMotor : FB_1011;
    M_Track_FWD : BOOL;  (* Motor track forward *)
    M_Track_REV : BOOL;  (* Motor track reverse *)
    Speed_Ref : INT;  (* Speed reference *)
    Inverter : FB_305;
    BeltUp_SA : BOOL;  (* Belt up semi automatic *)
    Comm : BOOL;
    Inverter_Track : FB_305;
    LS_Belt_Up : FB_101;
    LS_Belt_Down : FB_101;
    Beltmotor : FB_1011;
    Speed_Ref_Belt : INT;  (* Speed refeence belt *)
    Inverter_Belt : FB_305;
    M_Belt_FWD : BOOL;  (* Motor belt forward *)
    M_Belt_REV : BOOL;  (* Motor belt reverse *)
    Belt_Ref_Rev : BOOL;  (* Reference is reverse *)
    Belt_Ref_Fwd : BOOL;  (* Reference is forward *)
    ConditionsGlobal_Belt_Ok : BOOL;  (* Global conditions ok *)
    ConditionsFWD_Belt_Ok : BOOL;  (* Conditions forward ok *)
    COnditionsREV_Belt_Ok : BOOL;  (* Conditions reverse ok *)
    Track201HighSpeedStart : BOOL;  (* Start timer high speed *)
    TimerHighSpeed : _sTimer;  (* timer highspeed *)
    T_HighSpeed_Track201 : _sTimer;  (* Timer highspeed *)
    Track201Slow : BOOL;  (* track 201 slow *)
    Track202HighSpeedStart : BOOL;  (* Start timer high speed *)
    T_HighSpeed_Track202 : _sTimer;  (* Timer hig speed *)
    Track202Slow : BOOL;  (* Track 202 slow *)
    Semi_Automatic_Track : FB_307;
    Track_SA_FWD : BOOL;  (* Track semi automatic forward *)
    Track_SA_REV : BOOL;  (* Track semi automatic reverse *)
    Semi_Automatic_Belt : FB_307;
    Belt_SA_FWD : BOOL;  (* Belt semi automatic forward *)
    Belt_SA_REV : BOOL;  (* Belt semi automatic reverse *)
    T_BeltSpeedHigh : _sTimer;  (* Timer belt hig speed *)
    HB_TransferBufferOK : BOOL;
    Trans : BOOL;
    MachineInAlarm : BOOL;  (* Machine has an alarm *)
    T_Warning_BeltUp : _sTimer;
    T_Warning_BeltDown : _sTimer;
    HB_TransferBuffer201 : BOOL;
    HB_TransferBuffer202 : BOOL;
    ResetTrack : BOOL;  (* Reset track motor *)
    T_NoGrantLeave : _sTimer;  (* Timer no grant leave *)
    T_NoContainer : _sTimer;  (* Timer no container *)
END_VAR
VAR RETAIN
    Cyclus_st01 : BOOL;  (* Cycle: Instruction is correct. Start inbound *)
END_VAR
VAR
    Release : BOOL;  (* Clearance for outputs and cycle. EStop is OK and no alarms active. *)
    T_Power_OK : FB_101;
    T_Power_OK_DON : BOOL;  (* TImer power is on long enough *)
    Valve_Belt_Ref : BOOL;  (* Reference for belt valve. *)
    zz_Drew_Test : BOOL;
END_VAR
VAR_INPUT
    Enable : BOOL;
    EmergencyStopOk : BOOL;  (* Emergency stop OK *)
    MachineCode : UINT;  (* Machine code *)
    InverterStatus_Belt : ST_MX2\Status;  (* Inverterstatus *)
    InverterStatus_Track : ST_MX2\Status;  (* Inverterstatus *)
    Inputs : ST_FB_30051_Inputs;  (* IS_Track201 IS TRack 201; IS_Track202 IS track 202; IS_Present IS bench present; IS_PB_Run Pushbutton run motor; LS_BeltDown LS belt down; LS_BeltUp LS belt up *)
    Settings : ST_FB_30051_Settings;  (* TimeDelayON_IS201 Setting time delay on; TimeDelayOFF_IS201 Time delay off; TimeDelayON_IS202 Setting time delay on; TimeDelayOFF_IS202 Setting time delay off; TimeDelayON_LSTrackUp Setting time delay on; TimeDelayON_LSTrackDown Setting time delay on; TimeDelayON_ISPresent Setting time delay on; TimeDelayOFF_ISPresent Setting time delay off; TrackDirection Setting track direction; MAX_Run_Time Max run time; MinSpeed Minimal speed; Inverter_NodeNumber_Track Node number track; Inverter_Parameters_Track Inverter parameters; Inverter_Parameters_Belt Inverter parameters; MaxSpeed Max speed; UseInstructionTrack Use instruction for track; TimeHighSpeed Setting timer; MaxSpeedBelt Max sped belt; TimeHighSpeedBelt Time high speed *)
    CommIn101 : ST_Comm_Pipe_To_Track;
    CommIn201 : ST_Comm_Track_To_Track;
    CommIn202 : ST_Comm_Track_To_Track;
END_VAR
VAR_OUTPUT
    OUT_InverterCommands_Belt : ST_MX2\Command;  (* Inverter commands *)
    OUT_InverterCommands_Track : ST_MX2\Command;  (* Inverter commands *)
    OUT_InverterSpeed_Belt : INT;  (* Inverter speed *)
    OUT_InverterSpeed_Track : INT;  (* Inverter speed *)
    Outputs : ST_FB_30051_Outputs;
    CommOut_101 : ST_Comm_Track_To_Pipe;  (* StopOutbound Stop outbound *)
    CommOut_201 : ST_Comm_Track_To_Track;
    CommOut_202 : ST_Comm_Track_To_Track;
END_VAR
VAR_IN_OUT
    DatAControl : ST_DatAControl_Standard;  (* IN Dat A Control instruction; OUT.Instruction Dat A Control instruction out; OUT.Alarm04 Alarm word 4; IN.MachineMode Machine mode; IN.Settings.ResetAlarm Dat A Control Reset Alarm; IN.Settings.ResetCycle Dat A Control Reset Cycle; OUT.Alarm00 Alarm word 0; OUT.Alarm01 Alarm word 1; OUT.TotalDone Total done; OUT.Warning00 Warning word 0; OUT.Alarm02 Alarm word 2; OUT.CycleInformation Cycle information; OUT.Alarm03 Alarm word 3 *)
    Commands : ST_FB_30051_Commands;  (* Commands; BeltUp Commands belt up; BeltDown Commands belt down *)
    TransferBuffer : ST_TransferBuffer;  (* Transferbuffer *)
    Inverter_WriteParameters_Belt : BOOL;  (* Write parameters *)
    Inverter_WriteParameters_Track : BOOL;  (* Write parameters *)
    Inverter_WriteParametersDone_Belt : BOOL;  (* Write parameters done *)
    Inverter_WriteParametersDone_Track : BOOL;  (* Write parameters done *)
END_VAR
VAR_EXTERNAL
    Dummy : BOOL;
    ES_OK : BOOL;
END_VAR
VAR
    _e1 : R_TRIG;
    _t2 : BOOL;
    _t3 : BOOL;
    _e4 : R_TRIG;
    _e5 : R_TRIG;
    _p6 : BOOL;
    _p7 : BOOL;
    _e8 : R_TRIG;
    _e9 : R_TRIG;
    _t10 : BOOL;
    _t11 : BOOL;
    _t12 : BOOL;
    _p13 : BOOL;
    _t14 : BOOL;
    _p15 : BOOL;
    _p16 : BOOL;
    _t17 : BOOL;
END_VAR
(* ladder, written here as Structured Text *)

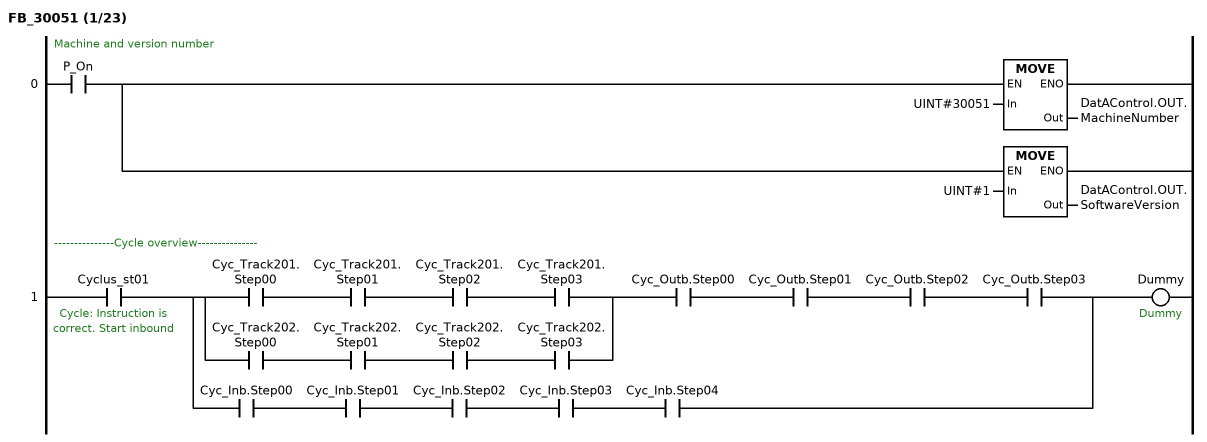
(* Rung 0: Machine and version number *)
IF P_On THEN
    DatAControl.OUT.MachineNumber := UINT#30051;
    DatAControl.OUT.SoftwareVersion := UINT#1;
END_IF;
(* Rung 1: ---------------Cycle overview--------------- *)
Dummy := Cyclus_st01 AND ((((Cyc_Track201.Step00 AND Cyc_Track201.Step01 AND Cyc_Track201.Step02 AND Cyc_Track201.Step03) OR (Cyc_Track202.Step00 AND Cyc_Track202.Step01 AND Cyc_Track202.Step02 AND Cyc_Track202.Step03)) AND Cyc_Outb.Step00 AND Cyc_Outb.Step01 AND Cyc_Outb.Step02 AND Cyc_Outb.Step03) OR (Cyc_Inb.Step00 AND Cyc_Inb.Step01 AND Cyc_Inb.Step02 AND Cyc_Inb.Step03 AND Cyc_Inb.Step04));

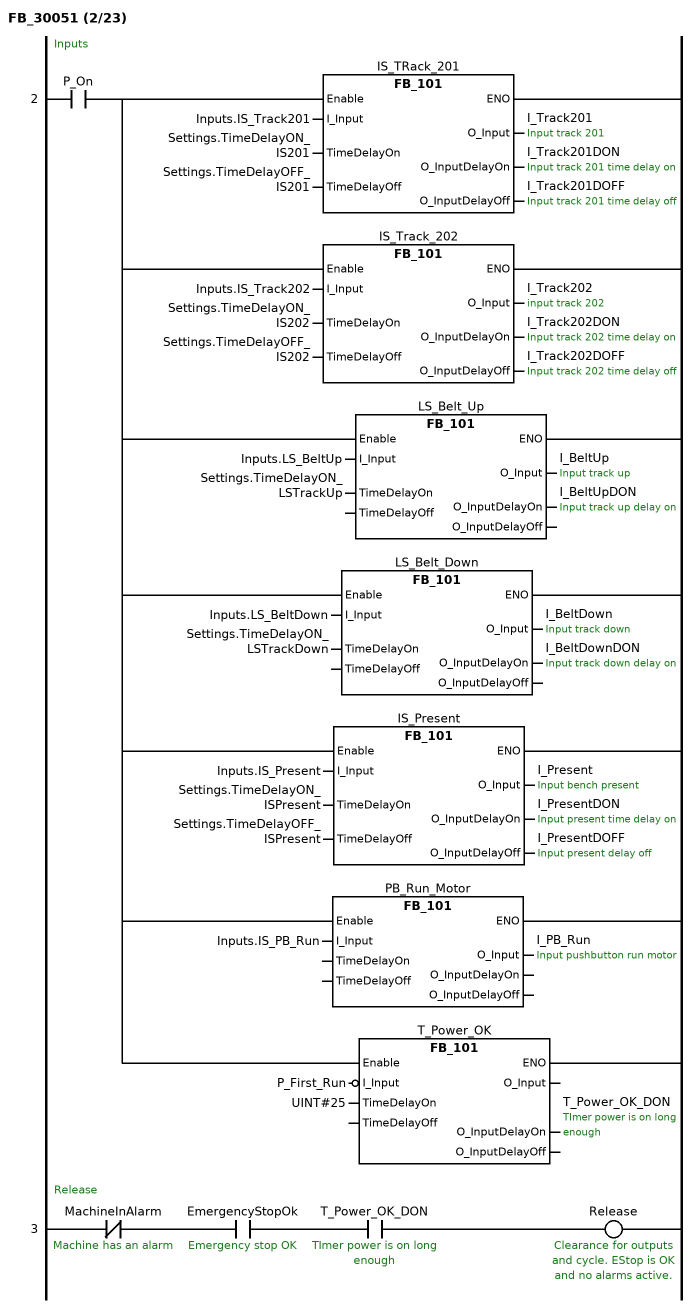
(* Rung 2: Inputs *)
IS_TRack_201(Enable := P_On, I_Input := Inputs.IS_Track201, TimeDelayOn := Settings.TimeDelayON_IS201, TimeDelayOff := Settings.TimeDelayOFF_IS201, O_Input => I_Track201, O_InputDelayOn => I_Track201DON, O_InputDelayOff => I_Track201DOFF);
IS_Track_202(Enable := P_On, I_Input := Inputs.IS_Track202, TimeDelayOn := Settings.TimeDelayON_IS202, TimeDelayOff := Settings.TimeDelayOFF_IS202, O_Input => I_Track202, O_InputDelayOn => I_Track202DON, O_InputDelayOff => I_Track202DOFF);
LS_Belt_Up(Enable := P_On, I_Input := Inputs.LS_BeltUp, TimeDelayOn := Settings.TimeDelayON_LSTrackUp, O_Input => I_BeltUp, O_InputDelayOn => I_BeltUpDON);
LS_Belt_Down(Enable := P_On, I_Input := Inputs.LS_BeltDown, TimeDelayOn := Settings.TimeDelayON_LSTrackDown, O_Input => I_BeltDown, O_InputDelayOn => I_BeltDownDON);
IS_Present(Enable := P_On, I_Input := Inputs.IS_Present, TimeDelayOn := Settings.TimeDelayON_ISPresent, TimeDelayOff := Settings.TimeDelayOFF_ISPresent, O_Input => I_Present, O_InputDelayOn => I_PresentDON, O_InputDelayOff => I_PresentDOFF);
PB_Run_Motor(Enable := P_On, I_Input := Inputs.IS_PB_Run, O_Input => I_PB_Run);
T_Power_OK(Enable := P_On, I_Input := NOT P_First_Run, TimeDelayOn := UINT#25, O_InputDelayOn => T_Power_OK_DON);
(* Rung 3: Release *)
Release := NOT MachineInAlarm AND EmergencyStopOk AND T_Power_OK_DON;

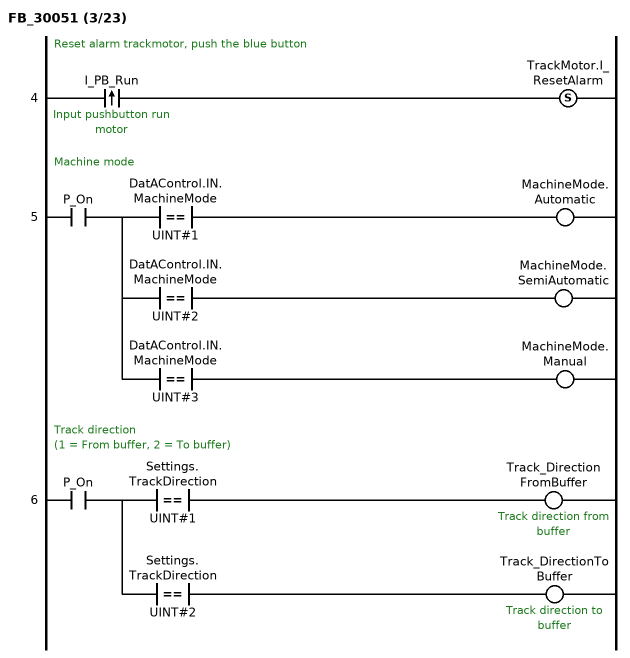
(* Rung 4: Reset alarm trackmotor, push the blue button *)
_e1(CLK := I_PB_Run);
IF _e1.Q THEN TrackMotor.I_ResetAlarm := TRUE; END_IF;
(* Rung 5: Machine mode *)
MachineMode.Automatic := P_On AND (DatAControl.IN.MachineMode = UINT#1);
MachineMode.SemiAutomatic := P_On AND (DatAControl.IN.MachineMode = UINT#2);
MachineMode.Manual := P_On AND (DatAControl.IN.MachineMode = UINT#3);
(* Rung 6: Track direction / (1 = From buffer, 2 = To buffer) *)
Track_DirectionFromBuffer := P_On AND (Settings.TrackDirection = UINT#1);
Track_DirectionToBuffer := P_On AND (Settings.TrackDirection = UINT#2);

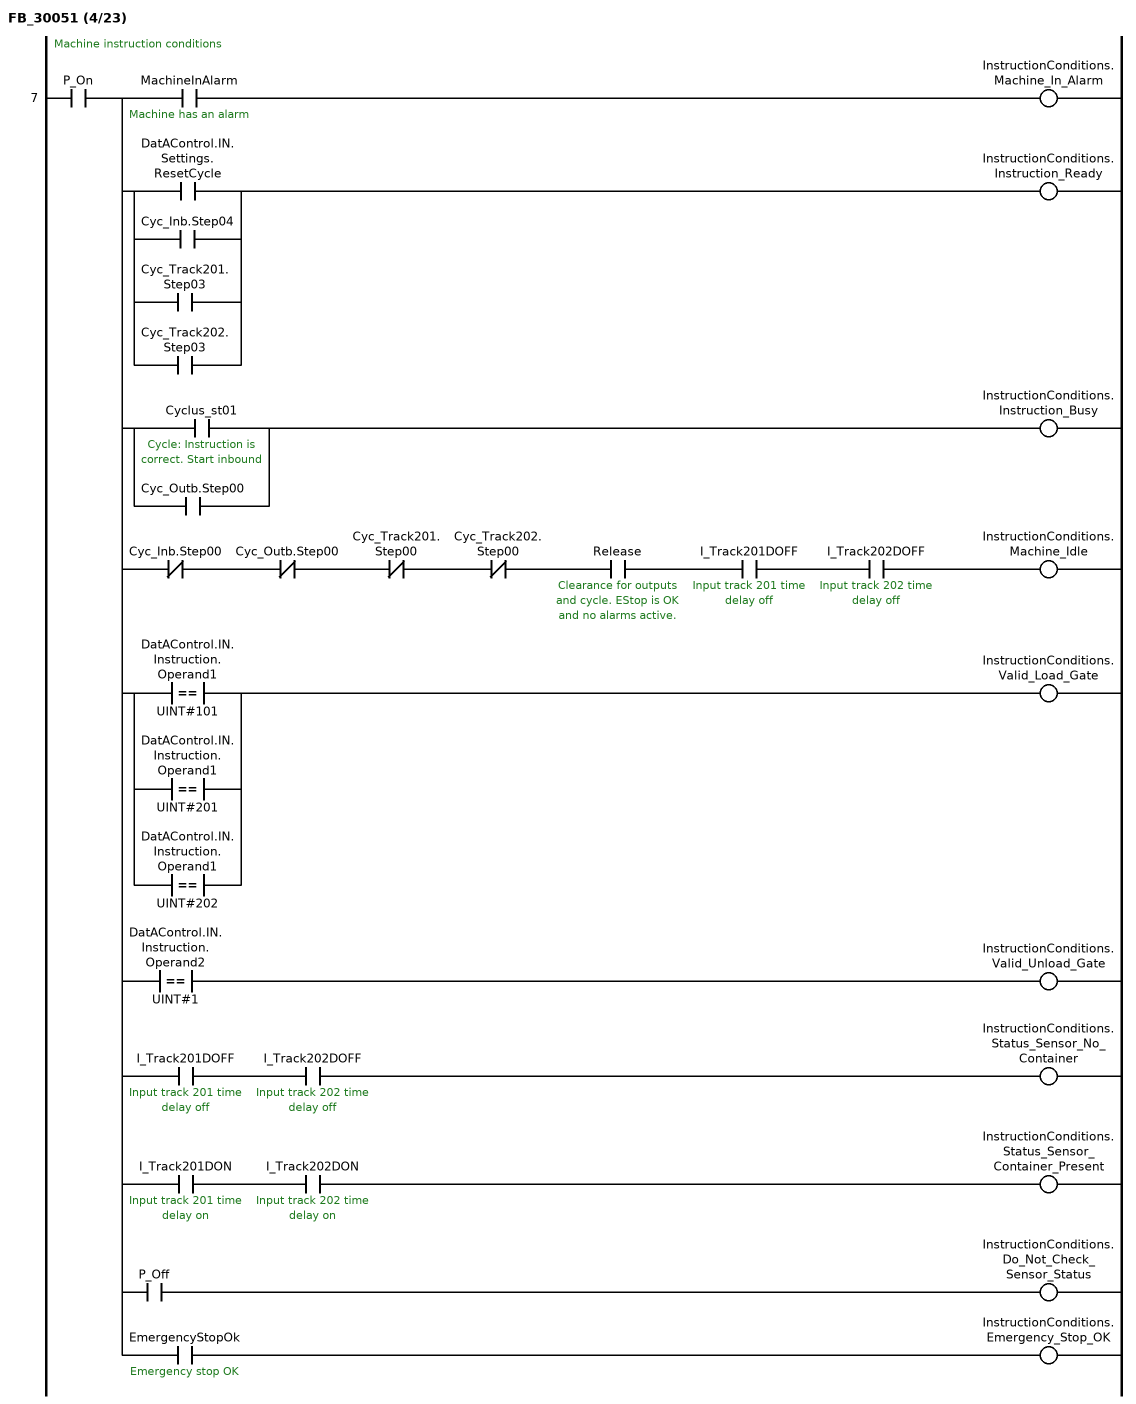
(* Rung 7: Machine instruction conditions *)
InstructionConditions.Machine_In_Alarm := P_On AND MachineInAlarm;
InstructionConditions.Instruction_Ready := P_On AND (DatAControl.IN.Settings.ResetCycle OR Cyc_Inb.Step04 OR Cyc_Track201.Step03 OR Cyc_Track202.Step03);
InstructionConditions.Instruction_Busy := P_On AND (Cyclus_st01 OR Cyc_Outb.Step00);
InstructionConditions.Machine_Idle := P_On AND NOT Cyc_Inb.Step00 AND NOT Cyc_Outb.Step00 AND NOT Cyc_Track201.Step00 AND NOT Cyc_Track202.Step00 AND Release AND I_Track201DOFF AND I_Track202DOFF;
InstructionConditions.Valid_Load_Gate := P_On AND ((DatAControl.IN.Instruction.Operand1 = UINT#101) OR (DatAControl.IN.Instruction.Operand1 = UINT#201) OR (DatAControl.IN.Instruction.Operand1 = UINT#202));
InstructionConditions.Valid_Unload_Gate := P_On AND (DatAControl.IN.Instruction.Operand2 = UINT#1);
InstructionConditions.Status_Sensor_No_Container := P_On AND I_Track201DOFF AND I_Track202DOFF;
InstructionConditions.Status_Sensor_Container_Present := P_On AND I_Track201DON AND I_Track202DON;
InstructionConditions.Do_Not_Check_Sensor_Status := P_On AND P_Off;
InstructionConditions.Emergency_Stop_OK := P_On AND EmergencyStopOk;

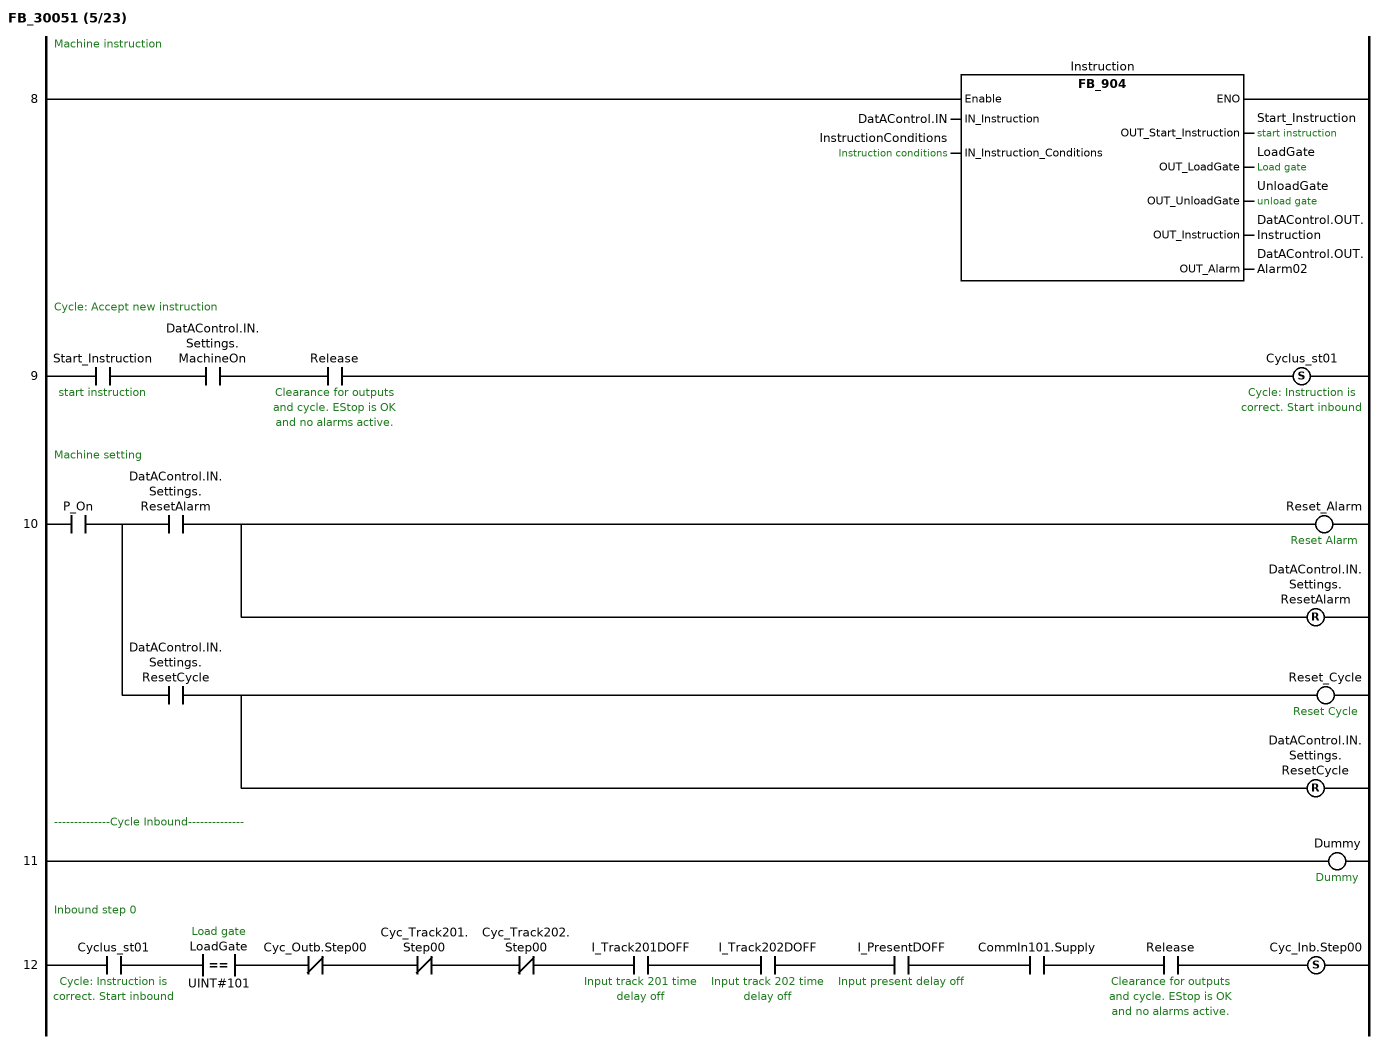
(* Rung 8: Machine instruction *)
Instruction(Enable := TRUE, IN_Instruction := DatAControl.IN, IN_Instruction_Conditions := InstructionConditions, OUT_Start_Instruction => Start_Instruction, OUT_LoadGate => LoadGate, OUT_UnloadGate => UnloadGate, OUT_Instruction => DatAControl.OUT.Instruction, OUT_Alarm => DatAControl.OUT.Alarm02);
(* Rung 9: Cycle: Accept new instruction *)
IF Start_Instruction AND DatAControl.IN.Settings.MachineOn AND Release THEN Cyclus_st01 := TRUE; END_IF;
(* Rung 10: Machine setting *)
Reset_Alarm := P_On AND DatAControl.IN.Settings.ResetAlarm;
IF P_On AND DatAControl.IN.Settings.ResetAlarm THEN DatAControl.IN.Settings.ResetAlarm := FALSE; END_IF;
Reset_Cycle := P_On AND DatAControl.IN.Settings.ResetCycle;
IF P_On AND DatAControl.IN.Settings.ResetCycle THEN DatAControl.IN.Settings.ResetCycle := FALSE; END_IF;
(* Rung 11: --------------Cycle Inbound-------------- *)
Dummy := TRUE;
(* Rung 12: Inbound step 0 *)
IF Cyclus_st01 AND (LoadGate = UINT#101) AND NOT Cyc_Outb.Step00 AND NOT Cyc_Track201.Step00 AND NOT Cyc_Track202.Step00 AND I_Track201DOFF AND I_Track202DOFF AND I_PresentDOFF AND CommIn101.Supply AND Release THEN
    Cyc_Inb.Step00 := TRUE;
END_IF;

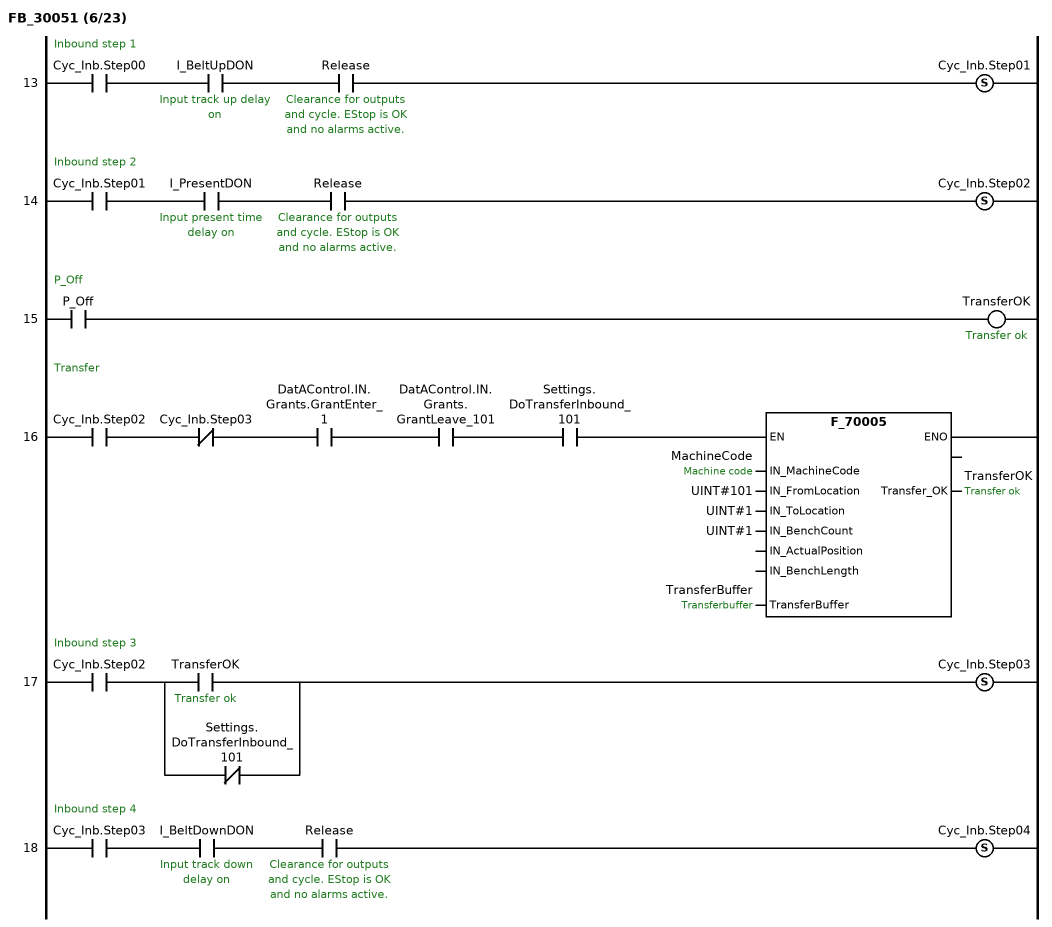
(* Rung 13: Inbound step 1 *)
IF Cyc_Inb.Step00 AND I_BeltUpDON AND Release THEN Cyc_Inb.Step01 := TRUE; END_IF;
(* Rung 14: Inbound step 2 *)
IF Cyc_Inb.Step01 AND I_PresentDON AND Release THEN Cyc_Inb.Step02 := TRUE; END_IF;
(* Rung 15: P_Off *)
TransferOK := P_Off;
(* Rung 16: Transfer *)
IF Cyc_Inb.Step02 AND NOT Cyc_Inb.Step03 AND DatAControl.IN.Grants.GrantEnter_1 AND DatAControl.IN.Grants.GrantLeave_101 AND Settings.DoTransferInbound_101 THEN
    F_70005(IN_MachineCode := MachineCode, IN_FromLocation := UINT#101, IN_ToLocation := UINT#1, IN_BenchCount := UINT#1, TransferBuffer := TransferBuffer, Transfer_OK => TransferOK);
END_IF;
(* Rung 17: Inbound step 3 *)
IF Cyc_Inb.Step02 AND (TransferOK OR NOT Settings.DoTransferInbound_101) THEN
    Cyc_Inb.Step03 := TRUE;
END_IF;
(* Rung 18: Inbound step 4 *)
IF Cyc_Inb.Step03 AND I_BeltDownDON AND Release THEN Cyc_Inb.Step04 := TRUE; END_IF;

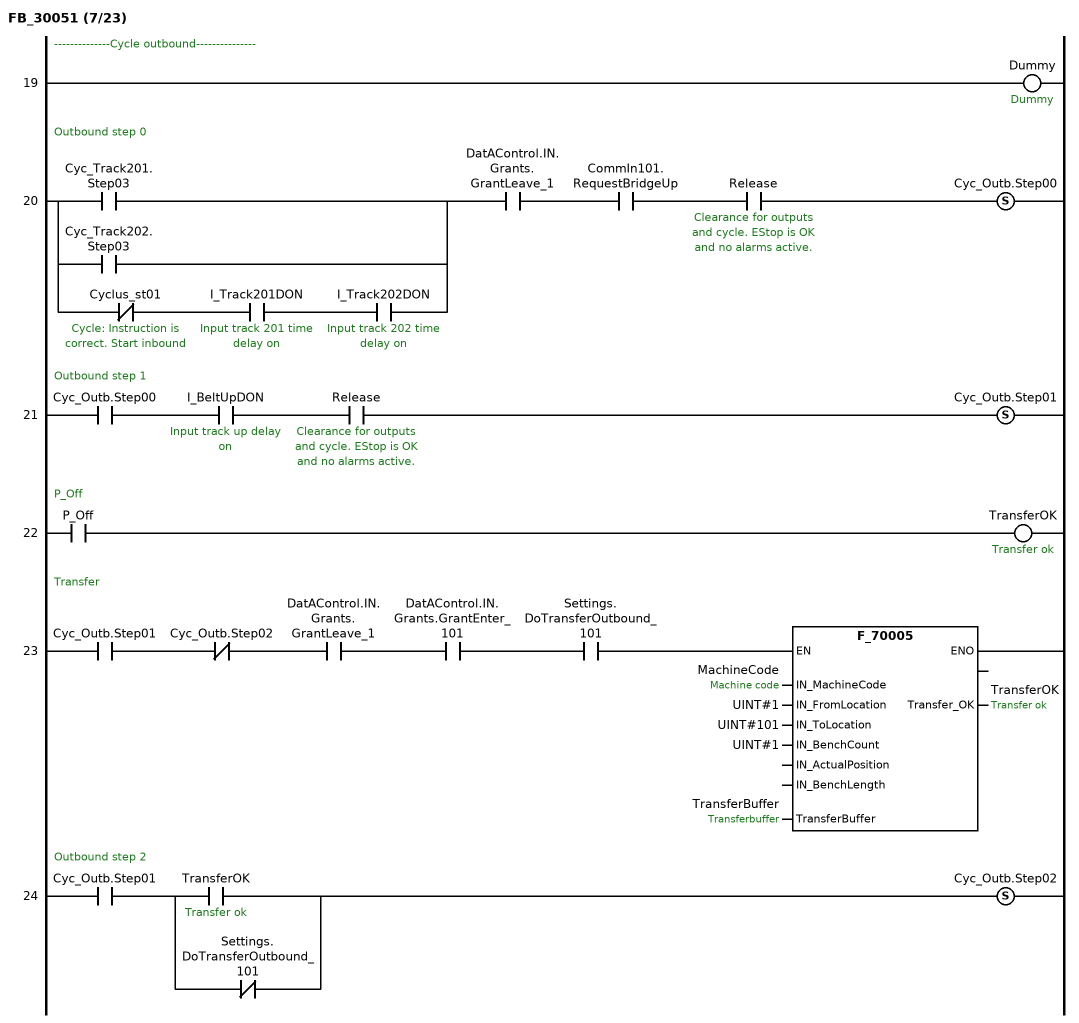
(* Rung 19: --------------Cycle outbound--------------- *)
Dummy := TRUE;
(* Rung 20: Outbound step 0 *)
IF (Cyc_Track201.Step03 OR Cyc_Track202.Step03 OR (NOT Cyclus_st01 AND I_Track201DON AND I_Track202DON)) AND DatAControl.IN.Grants.GrantLeave_1 AND CommIn101.RequestBridgeUp AND Release THEN
    Cyc_Outb.Step00 := TRUE;
END_IF;
(* Rung 21: Outbound step 1 *)
IF Cyc_Outb.Step00 AND I_BeltUpDON AND Release THEN Cyc_Outb.Step01 := TRUE; END_IF;
(* Rung 22: P_Off *)
TransferOK := P_Off;
(* Rung 23: Transfer *)
IF Cyc_Outb.Step01 AND NOT Cyc_Outb.Step02 AND DatAControl.IN.Grants.GrantLeave_1 AND DatAControl.IN.Grants.GrantEnter_101 AND Settings.DoTransferOutbound_101 THEN
    F_70005(IN_MachineCode := MachineCode, IN_FromLocation := UINT#1, IN_ToLocation := UINT#101, IN_BenchCount := UINT#1, TransferBuffer := TransferBuffer, Transfer_OK => TransferOK);
END_IF;
(* Rung 24: Outbound step 2 *)
IF Cyc_Outb.Step01 AND (TransferOK OR NOT Settings.DoTransferOutbound_101) THEN
    Cyc_Outb.Step02 := TRUE;
END_IF;

